// TwinCAT 3 PLC project tmo_optics
// Title: lcls-plc-tmo-optics
// Company: SLAC
// ProjectVersion: 0.0.0
// ProgramVersion: 3.1.4026.17
// CompilerDefines: K
// libraries:
//   LCLS General, * (SLAC)
//   lcls-twincat-common-components, * (SLAC)
//   lcls-twincat-optics, * (SLAC)
//   Tc2_MC2, * (Beckhoff Automation GmbH)
//   Tc2_SerialCom, * (Beckhoff Automation GmbH)
//   Tc2_Standard, * (Beckhoff Automation GmbH)
//   Tc2_System, * (Beckhoff Automation GmbH)
//   Tc2_Utilities, * (Beckhoff Automation GmbH)
//   Tc3_Module, * (Beckhoff Automation GmbH)
//   TcUnit, * (www.tcunit.org)
//   lcls-twincat-motion,4.2.0,SLAC
//   PMPS,3.4.1,SLAC - LCLS
// project tree:
//   DUTs/ ENUM_Si_B4C_Coating_States.TcDUT, E_HomeState.TcDUT (not stored)
//   GVLs/ GVL_COM_Buffers.TcGVL, GVL_M1K4.TcGVL, GVL_M1K4_Constants.TcGVL, GVL_M2K4_RTD.TcGVL, GVL_M2K4_Constants.TcGVL, GVL_M3K4_RTD.TcGVL, GVL_M3K4_Constants.TcGVL, GVL_M4K4_RTD.TcGVL, GVL_M5K4_RTD.TcGVL, GVL_PMPS.TcGVL, GVL_SerialIO.TcGVL
//   / PiezoDriver.TcTTO (not stored), PlcTask.TcTTO, SerialIO.TcTTO (not stored)
//   POUs/ FB_Offset_Coating_States.TcPOU, FB_KBO_Coating_States.TcPOU, Main.TcPOU, PRG_1_PlcTask.TcPOU, PRG_Environment.TcPOU, PRG_MR1K4_SOMS.TcPOU, PRG_MR2K4_KBO.TcPOU, PRG_MR3K4_KBO.TcPOU, PRG_MR4K4_KBO.TcPOU, PRG_MR5K4_KBO.TcPOU, PRG_PMPS.TcPOU, PRG_SL2K4_SCATTER.TcPOU, PRG_States.TcPOU, P_StripeProtections.TcPOU
//   POUs/Serial Comm/ PiezoSerial.TcPOU, P_Serial_Com.TcPOU
//   POUs/temp/ FB_SLITS.TcPOU
// real-time tasks:
//   TASK PlcTask: cycle T#10ms, priority 20, ADS port 350
//   TASK PiezoDriver: cycle T#1ms, priority 3, ADS port 351
//   TASK SerialIO: cycle T#2ms, priority 1, ADS port 352
// motion (NC):
//   TASK NC-Task 1 SAF: cycle T#2ms, priority 4, ADS port 501
//   TASK NC-Task 1 SVB: cycle T#10ms, priority 8, ADS port 511
//   AXIS M1K4-Yup (id 1)
//   AXIS M1K4-Ydwn (id 2)
//   AXIS M1K4-Xup (id 3)
//     General: UnitName=um
//     Dynamic: Acceleration=2000, Deceleration=2000, DelayTime=0.008
//     Velo: Maximum=1000
//     OtherSettings: AllowMotionCmdToSlave=true
//     encoder EncType=29
//       EncPara: ScaleFactorNumerator=0.001, Offset=-24000.3, MaxCount=#xffffffff
//         SoftEndMinControl: Enable=true, Range=-1500
//         SoftEndMaxControl: Enable=true, Range=1500
//         Inc: RefSoftSyncMask=#x0000ffff
//     drive DrvType=24
//       Analog: VeloReferenz=1220.703125, ScaleFactorActTorque=0.1
//       TimeComp: TaskDelayCycles=1
//     controller CtrType=2
//       CtrPara: PriorControlFactor=1
//         PosDiffControl: Range=100
//         PID: PosKp=50, PosExtKp=50, DeadBandPosition=0.4
//         Observer: BandWidth=20
//   AXIS M1K4-Xdwn (id 4)
//     General: UnitName=um
//     Dynamic: Acceleration=2000, Deceleration=2000, DelayTime=0.008
//     Velo: Maximum=1000
//     OtherSettings: AllowMotionCmdToSlave=true
//     encoder EncType=29
//       EncPara: ScaleFactorNumerator=0.001, Offset=-23999.4, MaxCount=#xffffffff
//         SoftEndMinControl: Enable=true, Range=-2000
//         SoftEndMaxControl: Enable=true, Range=2048.5
//         Inc: RefSoftSyncMask=#x0000ffff
//     drive DrvType=24
//       DrvPara: Inverse=true
//         Analog: VeloReferenz=1220.703125, ScaleFactorActTorque=0.1
//         TimeComp: TaskDelayCycles=1
//     controller CtrType=2
//       CtrPara: PriorControlFactor=1
//         PosDiffControl: Range=100
//         PID: PosKp=50, PosExtKp=50, DeadBandPosition=0.4
//         Observer: BandWidth=20
//   AXIS M1K4-Pitch (id 5)
//     General: UnitName=urad
//     Dynamic: Acceleration=390, Deceleration=390, DelayTime=0.008
//     Velo: Maximum=150
//     OtherSettings: AllowMotionCmdToSlave=true
//     encoder EncType=29
//       EncPara: ScaleFactorNumerator=0.001949317739, Offset=-19509, MaxCount=#xffffffff
//         FilterTime: TPos=0.2
//         SoftEndMinControl: Enable=true, Range=-60
//         SoftEndMaxControl: Enable=true, Range=180
//         Inc: RefSoftSyncMask=#x0000ffff
//     drive DrvType=24
//       Analog: VeloReferenz=371.8, ScaleFactorActTorque=0.1
//       TimeComp: TaskDelayCycles=1
//     controller CtrType=2
//       CtrPara: PriorControlFactor=1
//         PosDiffControl: Range=150
//         PID: PosKp=2, PosExtKp=1, DeadBandPosition=0.01
//         Observer: BandWidth=20
//   AXIS M1K4-Bender (id 6)
//     General: UnitName=um
//     Dynamic: Acceleration=100, Deceleration=100, DelayTime=0.008
//     Velo: Maximum=150
//     OtherSettings: AllowMotionCmdToSlave=true
//     encoder EncType=29
//       EncPara: ScaleFactorNumerator=0.001, MaxCount=#xffffffff
//         Inc: RefSoftSyncMask=#x0000ffff
//     drive DrvType=24
//       Analog: VeloReferenz=195.3125, ScaleFactorActTorque=0.1
//       TimeComp: TaskDelayCycles=1
//     controller CtrType=2
//       CtrPara: PriorControlFactor=1
//         PID: PosKp=10, PosExtKp=1, DeadBandPosition=0.04
//         Observer: BandWidth=20
//   AXIS M2K4-X (id 7)
//     Dynamic: AccelerationMaximum=100, DecelerationMaximum=100, Acceleration=100, Deceleration=100, DelayTime=0.008
//     Velo: Maximum=20
//     OtherSettings: AllowMotionCmdToSlave=true
//     encoder EncType=29
//       EncPara: ScaleFactorNumerator=5e-06, Offset=-30.6825, MaxCount=#xffffffff, ReferenceSystem=1
//         SoftEndMinControl: Enable=true, Range=0.2
//         SoftEndMaxControl: Enable=true, Range=2.1
//         Inc: RefSoftSyncMask=#x0000ffff
//     drive DrvType=24
//       DrvPara: Inverse=true
//         Analog: VeloReferenz=20, ScaleFactorActTorque=0.1
//         TimeComp: TaskDelayCycles=1
//     controller CtrType=2
//       CtrPara: PriorControlFactor=1
//         PosDiffControl: Range=0.1
//         PID: DeadBandPosition=0.001
//         Observer: BandWidth=20
//   AXIS M2K4-Y (id 8)
//     Dynamic: AccelerationMaximum=10, DecelerationMaximum=10, Acceleration=10, Deceleration=10, Jerk=15, DelayTime=0.008
//     Velo: Maximum=1.25
//     OtherSettings: AllowMotionCmdToSlave=true
//     encoder EncType=29
//       EncPara: ScaleFactorNumerator=5e-06, Offset=-30.18, MaxCount=#xffffffff, ReferenceSystem=1
//         SoftEndMinControl: Enable=true, Range=-12.5
//         SoftEndMaxControl: Enable=true, Range=13.39
//         Inc: RefSoftSyncMask=#x0000ffff
//     drive DrvType=24
//       DrvPara: Inverse=true
//         Analog: VeloReferenz=1.25, ScaleFactorActTorque=0.1
//         TimeComp: TaskDelayCycles=1
//     controller CtrType=2
//       CtrPara: PriorControlFactor=1
//         PosDiffControl: Range=0.1
//         PID: DeadBandPosition=0.001
//         Observer: BandWidth=20
//   AXIS M2K4-rY (id 9)
//     General: UnitName=urad
//     Dynamic: AccelerationMaximum=400, DecelerationMaximum=400, Acceleration=400, Deceleration=400, Jerk=1200, DelayTime=0.008
//     Velo: Maximum=166.67
//     OtherSettings: AllowMotionCmdToSlave=true
//     encoder EncType=29
//       EncPara: ScaleFactorNumerator=0.005348, Offset=-194502.025, MaxCount=#xffffffff, ReferenceSystem=1
//         FilterTime: TPos=0.01
//         SoftEndMinControl: Enable=true, Range=14370
//         SoftEndMaxControl: Enable=true, Range=14850
//         Inc: RefSoftSyncMask=#x0000ffff
//     drive DrvType=24
//       Analog: VeloReferenz=166.67, ScaleFactorActTorque=0.1
//       TimeComp: TaskDelayCycles=1
//     controller CtrType=2
//       CtrPara: PriorControlFactor=1
//         PosDiffControl: Range=40
//         PID: PosKp=0.5, DeadBandPosition=0.01
//         Observer: BandWidth=20
//   AXIS M2K4-BEND-US (id 10)
//     Dynamic: AccelerationMaximum=0.6, DecelerationMaximum=0.6, Acceleration=0.6, Deceleration=0.6, Jerk=1.2, DelayTime=0.008
//     Velo: Maximum=0.1
//     OtherSettings: AllowMotionCmdToSlave=true
//     encoder EncType=29
//       EncPara: ScaleFactorNumerator=1e-06, MaxCount=#xffffffff, ReferenceSystem=1
//         SoftEndMinControl: Enable=true, Range=6.4549
//         SoftEndMaxControl: Enable=true, Range=16.0941
//         Inc: RefSoftSyncMask=#x0000ffff
//     drive DrvType=24
//       DrvPara: Inverse=true
//         Analog: VeloReferenz=0.1, ScaleFactorActTorque=0.1
//         TimeComp: TaskDelayCycles=1
//     controller CtrType=2
//       CtrPara: PriorControlFactor=1
//         PosDiffControl: Range=0.2
//         PID: PosKp=15, PosExtKp=1, DeadBandPosition=0.0002
//         Observer: BandWidth=20
//   AXIS M2K4-BEND-DS (id 11)
//     Dynamic: AccelerationMaximum=0.6, DecelerationMaximum=0.6, Acceleration=0.6, Deceleration=0.6, Jerk=1.2, DelayTime=0.008
//     Velo: Maximum=0.1
//     OtherSettings: AllowMotionCmdToSlave=true
//     encoder EncType=29
//       EncPara: ScaleFactorNumerator=1e-06, MaxCount=#xffffffff, ReferenceSystem=1
//         SoftEndMinControl: Enable=true, Range=10.5742
//         SoftEndMaxControl: Enable=true, Range=22.2169
//         Inc: RefSoftSyncMask=#x0000ffff
//     drive DrvType=24
//       DrvPara: Inverse=true
//         Analog: VeloReferenz=0.1, ScaleFactorActTorque=0.1
//         TimeComp: TaskDelayCycles=1
//     controller CtrType=2
//       CtrPara: PriorControlFactor=1
//         PosDiffControl: Range=0.2
//         PID: PosKp=15, PosExtKp=1, DeadBandPosition=0.0002
//         Observer: BandWidth=20
//   AXIS M3K4-X (id 12)
//     Dynamic: AccelerationMaximum=100, DecelerationMaximum=100, Acceleration=100, Deceleration=100, DelayTime=0.008
//     Velo: Maximum=20
//     OtherSettings: AllowMotionCmdToSlave=true
//     encoder EncType=29
//       EncPara: ScaleFactorNumerator=5e-06, Offset=-31.1, MaxCount=#xffffffff, ReferenceSystem=1
//         SoftEndMinControl: Enable=true, Range=-10.179
//         SoftEndMaxControl: Enable=true, Range=12.0995
//         Inc: RefSoftSyncMask=#x0000ffff
//     drive DrvType=24
//       DrvPara: Inverse=true
//         Analog: VeloReferenz=20, ScaleFactorActTorque=0.1
//         TimeComp: TaskDelayCycles=1
//     controller CtrType=2
//       CtrPara: PriorControlFactor=1
//         PosDiffControl: Range=0.1
//         PID: DeadBandPosition=0.001
//         Observer: BandWidth=20
//   AXIS M3K4-Y (id 13)
//     Dynamic: AccelerationMaximum=10, DecelerationMaximum=10, Acceleration=10, Deceleration=10, Jerk=15, DelayTime=0.008
//     Velo: Maximum=1.25
//     OtherSettings: AllowMotionCmdToSlave=true
//     encoder EncType=29
//       EncPara: ScaleFactorNumerator=5e-06, Offset=-29.68, MaxCount=#xffffffff, ReferenceSystem=1
//         SoftEndMinControl: Enable=true, Range=0.25
//         SoftEndMaxControl: Enable=true, Range=2.15
//         Inc: RefSoftSyncMask=#x0000ffff
//     drive DrvType=24
//       DrvPara: Inverse=true
//         Analog: VeloReferenz=1.25, ScaleFactorActTorque=0.1
//         TimeComp: TaskDelayCycles=1
//     controller CtrType=2
//       CtrPara: PriorControlFactor=1
//         PosDiffControl: Range=0.1
//         PID: DeadBandPosition=0.001
//         Observer: BandWidth=20
//   AXIS M3K4-rX (id 14)
//     General: UnitName=urad
//     Dynamic: AccelerationMaximum=300, DecelerationMaximum=300, Acceleration=300, Deceleration=300, Jerk=900, DelayTime=0.008
//     Velo: Maximum=140.84
//     OtherSettings: AllowMotionCmdToSlave=true
//     encoder EncType=29
//       EncPara: ScaleFactorNumerator=0.002577, Offset=-136547, MaxCount=#xffffffff, ReferenceSystem=1
//         FilterTime: TPos=0.01
//         SoftEndMinControl: Enable=true, Range=-12560
//         SoftEndMaxControl: Enable=true, Range=-12090
//         Inc: RefSoftSyncMask=#x0000ffff
//     drive DrvType=24
//       Analog: VeloReferenz=140.84, ScaleFactorActTorque=0.1
//       TimeComp: TaskDelayCycles=1
//     controller CtrType=2
//       CtrPara: PriorControlFactor=1
//         PosDiffControl: Range=10
//         PID: PosKp=0.5, DeadBandPosition=0.01
//         Observer: BandWidth=20
//   AXIS M3K4-BEND-US (id 15)
//     Dynamic: AccelerationMaximum=0.6, DecelerationMaximum=0.6, Acceleration=0.6, Deceleration=0.6, Jerk=1.2, DelayTime=0.008
//     Velo: Maximum=0.1
//     OtherSettings: AllowMotionCmdToSlave=true
//     encoder EncType=29
//       EncPara: ScaleFactorNumerator=1e-06, MaxCount=#xffffffff, ReferenceSystem=1
//         SoftEndMinControl: Enable=true, Range=12.5315
//         SoftEndMaxControl: Enable=true, Range=22.979
//         Inc: RefSoftSyncMask=#x0000ffff
//     drive DrvType=24
//       DrvPara: Inverse=true
//         Analog: VeloReferenz=0.1, ScaleFactorActTorque=0.1
//         TimeComp: TaskDelayCycles=1
//     controller CtrType=2
//       CtrPara: PriorControlFactor=1
//         PosDiffControl: Range=0.2
//         PID: PosKp=15, PosExtKp=1, DeadBandPosition=0.0002
//         Observer: BandWidth=20
//   AXIS M3K4-BEND-DS (id 16)
//     Dynamic: AccelerationMaximum=0.6, DecelerationMaximum=0.6, Acceleration=0.6, Deceleration=0.6, Jerk=1.2, DelayTime=0.008
//     Velo: Maximum=0.1
//     OtherSettings: AllowMotionCmdToSlave=true
//     encoder EncType=29
//       EncPara: ScaleFactorNumerator=1e-06, MaxCount=#xffffffff, ReferenceSystem=1
//         SoftEndMinControl: Enable=true, Range=8.0419
//         SoftEndMaxControl: Enable=true, Range=22.8443
//         Inc: RefSoftSyncMask=#x0000ffff
//     drive DrvType=24
//       DrvPara: Inverse=true
//         Analog: VeloReferenz=0.1, ScaleFactorActTorque=0.1
//         TimeComp: TaskDelayCycles=1
//     controller CtrType=2
//       CtrPara: PriorControlFactor=1
//         PosDiffControl: Range=0.2
//         PID: PosKp=15, PosExtKp=1, DeadBandPosition=0.0002
//         Observer: BandWidth=20
//   AXIS M4K4 X (id 17)
//     Dynamic: AccelerationMaximum=100, DecelerationMaximum=100, Acceleration=100, Deceleration=100, DelayTime=0.008
//     Velo: Maximum=0.3
//     OtherSettings: AllowMotionCmdToSlave=true
//     encoder EncType=29
//       EncPara: ScaleFactorNumerator=5e-06, Offset=-28.961399, MaxCount=#xffffffff, ReferenceSystem=1
//         SoftEndMinControl: Range=-11.2
//         SoftEndMaxControl: Range=13.2
//         Inc: RefSoftSyncMask=#x0000ffff
//     drive DrvType=24
//       DrvPara: Inverse=true
//         Analog: VeloReferenz=20, ScaleFactorActTorque=0.1
//         TimeComp: TaskDelayCycles=1
//     controller CtrType=2
//       CtrPara: PriorControlFactor=1
//         PosDiffControl: Range=0.2
//         PID: DeadBandPosition=0.001
//         Observer: BandWidth=20
//   AXIS M4K4 Y (id 18)
//     Dynamic: AccelerationMaximum=100, DecelerationMaximum=100, Acceleration=100, Deceleration=100, DelayTime=0.008
//     Velo: Maximum=0.2
//     OtherSettings: AllowMotionCmdToSlave=true
//     encoder EncType=29
//       EncPara: ScaleFactorNumerator=5e-06, Offset=-30.3992, MaxCount=#xffffffff, ReferenceSystem=1
//         SoftEndMinControl: Enable=true, Range=-0.5
//         SoftEndMaxControl: Enable=true, Range=1.25
//         Inc: RefSoftSyncMask=#x0000ffff
//     drive DrvType=24
//       DrvPara: Inverse=true
//         Analog: VeloReferenz=1.25, ScaleFactorActTorque=0.1
//         TimeComp: TaskDelayCycles=1
//     controller CtrType=2
//       CtrPara: PriorControlFactor=1
//         PosDiffControl: Range=0.2
//         PID: PosKp=3, DeadBandPosition=0.001
//         Observer: BandWidth=20
//   AXIS M4K4 Z (id 19)
//     Dynamic: AccelerationMaximum=100, DecelerationMaximum=100, Acceleration=100, Deceleration=100, DelayTime=0.008
//     Velo: Maximum=0.2
//     OtherSettings: AllowMotionCmdToSlave=true
//     encoder EncType=29
//       EncPara: ScaleFactorNumerator=5e-06, Offset=-21445.3535, MaxCount=#xffffffff, ReferenceSystem=1
//         SoftEndMinControl: Enable=true, Range=-1.5
//         SoftEndMaxControl: Enable=true, Range=0.85
//         Inc: RefSoftSyncMask=#x0000ffff
//     drive DrvType=24
//       DrvPara: Inverse=true
//         Analog: VeloReferenz=1.25, ScaleFactorActTorque=0.1
//         TimeComp: TaskDelayCycles=1
//     controller CtrType=2
//       CtrPara: PriorControlFactor=1
//         PosDiffControl: Range=0.2
//         PID: PosKp=2, DeadBandPosition=0.01
//         Observer: BandWidth=20
//   AXIS M4K4 rX (id 20)
//     General: UnitName=urad
//     Dynamic: AccelerationMaximum=100, DecelerationMaximum=100, Acceleration=100, Deceleration=100, DelayTime=0.008
//     Velo: Maximum=50
//     OtherSettings: AllowMotionCmdToSlave=true
//     encoder EncType=29
//       EncPara: ScaleFactorNumerator=0.0025826, Offset=-132192.8499, MaxCount=#xffffffff, ReferenceSystem=1
//         FilterTime: TPos=0.2
//         SoftEndMinControl: Enable=true, Range=-300
//         SoftEndMaxControl: Enable=true, Range=35
//         Inc: RefSoftSyncMask=#x0000ffff
//     drive DrvType=24
//       Analog: VeloReferenz=140.69, ScaleFactorActTorque=0.1
//       TimeComp: TaskDelayCycles=1
//     controller CtrType=2
//       CtrPara: PriorControlFactor=1
//         PosDiffControl: Range=10
//         PID: PosExtKp=4, DeadBandPosition=0.01
//         Observer: BandWidth=20
//   AXIS M5K4 X (id 21)
//     Dynamic: AccelerationMaximum=100, DecelerationMaximum=100, Acceleration=100, Deceleration=100, DelayTime=0.008
//     Velo: Maximum=0.2
//     OtherSettings: AllowMotionCmdToSlave=true
//     encoder EncType=29
//       EncPara: ScaleFactorNumerator=5e-06, Offset=-29.80379, MaxCount=#xffffffff, ReferenceSystem=1
//         SoftEndMinControl: Enable=true, Range=-2.3
//         SoftEndMaxControl: Enable=true, Range=-0.37
//         Inc: RefSoftSyncMask=#x0000ffff
//     drive DrvType=24
//       DrvPara: Inverse=true
//         Analog: VeloReferenz=20, ScaleFactorActTorque=0.1
//         TimeComp: TaskDelayCycles=1
//     controller CtrType=2
//       CtrPara: PriorControlFactor=1
//         PosDiffControl: Range=0.2
//         PID: DeadBandPosition=0.001
//         Observer: BandWidth=20
//   AXIS M5K4 Y (id 22)
//     Dynamic: AccelerationMaximum=100, DecelerationMaximum=100, Acceleration=100, Deceleration=100, DelayTime=0.008
//     Velo: Maximum=0.3
//     OtherSettings: AllowMotionCmdToSlave=true
//     encoder EncType=29
//       EncPara: ScaleFactorNumerator=5e-06, Offset=-29.7766, MaxCount=#xffffffff, ReferenceSystem=1
//         SoftEndMinControl: Range=-12.3
//         SoftEndMaxControl: Range=12.33
//         Inc: RefSoftSyncMask=#x0000ffff
//     drive DrvType=24
//       DrvPara: Inverse=true
//         Analog: VeloReferenz=1.25, ScaleFactorActTorque=0.1
//         TimeComp: TaskDelayCycles=1
//     controller CtrType=2
//       CtrPara: PriorControlFactor=1
//         PosDiffControl: Range=0.2
//         PID: DeadBandPosition=0.001
//         Observer: BandWidth=20
//   AXIS M5K4 Z (id 23)
//     Dynamic: AccelerationMaximum=100, DecelerationMaximum=100, Acceleration=100, Deceleration=100, DelayTime=0.008
//     Velo: Maximum=0.2
//     OtherSettings: AllowMotionCmdToSlave=true
//     encoder EncType=29
//       EncPara: ScaleFactorNumerator=5e-06, Offset=-21444.5039, MaxCount=#xffffffff, ReferenceSystem=1
//         SoftEndMinControl: Enable=true, Range=-0.69
//         SoftEndMaxControl: Enable=true, Range=1.02
//         Inc: RefSoftSyncMask=#x0000ffff
//     drive DrvType=24
//       DrvPara: Inverse=true
//         Analog: VeloReferenz=1.25, ScaleFactorActTorque=0.1
//         TimeComp: TaskDelayCycles=1
//     controller CtrType=2
//       CtrPara: PriorControlFactor=1
//         PosDiffControl: Range=0.2
//         PID: PosExtVelo=1, DeadBandPosition=0.01
//         Observer: BandWidth=20
//   AXIS M5K4 rY (id 24)
//     General: UnitName=urad
//     Dynamic: AccelerationMaximum=100, DecelerationMaximum=100, Acceleration=100, Deceleration=100, DelayTime=0.008
//     Velo: Maximum=50
//     OtherSettings: AllowMotionCmdToSlave=true
//     encoder EncType=29
//       EncPara: ScaleFactorNumerator=0.00504, Offset=-198169.78, MaxCount=#xffffffff, ReferenceSystem=1
//         FilterTime: TPos=0.2
//         SoftEndMinControl: Enable=true, Range=-260
//         SoftEndMaxControl: Enable=true, Range=200
//         Inc: RefSoftSyncMask=#x0000ffff
//     drive DrvType=24
//       Analog: VeloReferenz=192.31, ScaleFactorActTorque=0.1
//       TimeComp: TaskDelayCycles=1
//     controller CtrType=2
//       CtrPara: PriorControlFactor=1
//         PosDiffControl: Range=10
//         PID: PosKp=2, PosExtKp=10, DeadBandPosition=0.01
//         Observer: BandWidth=20
//   AXIS SL2K4_TOP (id 25)
//     Dynamic: AccelerationMaximum=0.25, DecelerationMaximum=0.25, Acceleration=0.25, Deceleration=0.25, Jerk=0.4
//     Velo: RefSearch=0.05, RefSync=0.025, SlowManual=0.1, FastManual=0.1, Fast=3, Maximum=0.5
//     PositionAreaControl: Enable=false
//     TargetPosControl: Range=0.01
//     OtherSettings: AllowMotionCmdToSlave=true, PulseDistancePos=0.005, PulseDistanceNeg=0.005
//     encoder EncType=4
//       EncPara: ScaleFactorNumerator=1e-06, Inverse=true, MaxCount=#xffffffff
//         SoftEndMinControl: Enable=true, Range=-0.1
//         SoftEndMaxControl: Enable=true, Range=4.35
//         Inc: RefSoftSyncMask=#x0000ffff
//     drive DrvType=24
//       DrvPara: Inverse=true
//         Analog: VeloReferenz=3, TorqueSetpointScale=10, ScaleFactorActTorque=0.1
//         TimeComp: TaskDelayCycles=1
//     controller CtrType=1
//       CtrPara: PriorControlFactor=1
//         PosDiffControl: Range=0.2
//         Observer: BandWidth=20
//   AXIS SL2K4_BOTTOM (id 26)
//     Dynamic: AccelerationMaximum=0.25, DecelerationMaximum=0.25, Acceleration=0.25, Deceleration=0.25, Jerk=0.4
//     Velo: RefSearch=0.05, RefSync=0.025, SlowManual=0.1, FastManual=0.1, Maximum=0.5
//     PositionAreaControl: Enable=false
//     TargetPosControl: Range=0.01
//     OtherSettings: AllowMotionCmdToSlave=true, PulseDistancePos=0.005, PulseDistanceNeg=0.005
//     encoder EncType=4
//       EncPara: ScaleFactorNumerator=1e-06, MaxCount=#xffffffff
//         SoftEndMinControl: Enable=true, Range=-4.6
//         SoftEndMaxControl: Enable=true, Range=-0.4
//         Inc: RefSoftSyncMask=#x0000ffff
//     drive DrvType=24
//       Analog: VeloReferenz=3, TorqueSetpointScale=10, ScaleFactorActTorque=0.1
//       TimeComp: TaskDelayCycles=1
//     controller CtrType=1
//       CtrPara: PriorControlFactor=1
//         PosDiffControl: Range=0.2
//         Observer: BandWidth=20
//   AXIS SL2K4_NORTH (id 27)
//     Dynamic: AccelerationMaximum=0.25, DecelerationMaximum=0.25, Acceleration=0.25, Deceleration=0.25, Jerk=0.4
//     Velo: RefSearch=0.05, RefSync=0.025, SlowManual=0.1, FastManual=0.1, Maximum=0.5
//     OtherSettings: AllowMotionCmdToSlave=true, PulseDistancePos=0.005, PulseDistanceNeg=0.005
//     encoder EncType=4
//       EncPara: ScaleFactorNumerator=1e-06, Inverse=true, MaxCount=#xffffffff
//         SoftEndMinControl: Enable=true, Range=0.3
//         SoftEndMaxControl: Enable=true, Range=4.35
//         Inc: RefSoftSyncMask=#x0000ffff
//     drive DrvType=24
//       DrvPara: Inverse=true
//         Analog: VeloReferenz=3, TorqueSetpointScale=10, ScaleFactorActTorque=0.1
//         TimeComp: TaskDelayCycles=1
//     controller CtrType=1
//       CtrPara: PriorControlFactor=1
//         PosDiffControl: Range=0.2
//         Observer: BandWidth=20
//   AXIS SL2K4_SOUTH (id 28)
//     Dynamic: AccelerationMaximum=0.25, DecelerationMaximum=0.25, Acceleration=0.25, Deceleration=0.25, Jerk=0.4
//     Velo: RefSearch=0.05, RefSync=0.025, SlowManual=0.1, FastManual=0.1, Maximum=0.5
//     TargetPosControl: Range=0.01
//     OtherSettings: AllowMotionCmdToSlave=true, PulseDistancePos=0.005, PulseDistanceNeg=0.005
//     encoder EncType=4
//       EncPara: ScaleFactorNumerator=1e-06, MaxCount=#xffffffff
//         SoftEndMinControl: Enable=true, Range=-4.5
//         SoftEndMaxControl: Enable=true, Range=-0.3
//         Inc: RefSoftSyncMask=#x0000ffff
//     drive DrvType=24
//       Analog: VeloReferenz=3, TorqueSetpointScale=10, ScaleFactorActTorque=0.1
//       TimeComp: TaskDelayCycles=1
//     controller CtrType=1
//       CtrPara: PriorControlFactor=1
//         PosDiffControl: Range=0.2
//         Observer: BandWidth=20
// I/O:
//   DEVICE Device 1 (EtherCAT), AmsNetId 172.21.92.63.2.1
//     Term 1 (EK1200)
// variable links:
//   Axes/M4K4 X <-> Device 1 (EtherCAT)/Term 1 (EK1200)/Term 39 (EK1122)/Term 94 (EK1100)/EL5042_M4K4X_M4K4Y
//     Enc/Inputs/In/nComState @bit 1 <-> WcState/InputToggle
//     Enc/Inputs/In/nComState <-> WcState/WcState
//     Enc/Inputs/In/nDataIn1 <-> FB Inputs Channel 1/Position
//     Enc/Inputs/In/nState1 @bit 12 <-> FB Inputs Channel 1/Status/Diag
//     Enc/Inputs/In/nState1 @bit 1 <-> FB Inputs Channel 1/Status/Error
//     Enc/Inputs/In/nState1 @bit 14 <-> FB Inputs Channel 1/Status/Input cycle counter
//     Enc/Inputs/In/nState1 @bit 2 <-> FB Inputs Channel 1/Status/Ready
//     Enc/Inputs/In/nState1 @bit 13 <-> FB Inputs Channel 1/Status/TxPDO State
//     Enc/Inputs/In/nState1 <-> FB Inputs Channel 1/Status/Warning
//   Axes/M4K4 X <-> Device 1 (EtherCAT)/Term 1 (EK1200)/Term 39 (EK1122)/Term 94 (EK1100)/EL7041-0052_M4K4X
//     Drive/Inputs/In/nState1 @bit 3 <-> STM Status/Status/Error
//     Drive/Inputs/In/nState1 @bit 5 <-> STM Status/Status/Moving negative
//     Drive/Inputs/In/nState1 @bit 4 <-> STM Status/Status/Moving positive
//     Drive/Inputs/In/nState1 @bit 1 <-> STM Status/Status/Ready
//     Drive/Inputs/In/nState1 <-> STM Status/Status/Ready to enable
//     Drive/Inputs/In/nState1 @bit 6 <-> STM Status/Status/Torque reduced
//     Drive/Inputs/In/nState1 @bit 2 <-> STM Status/Status/Warning
//     Drive/Inputs/In/nState2 @bit 3 <-> STM Status/Status/Digital input 1
//     Drive/Inputs/In/nState2 @bit 4 <-> STM Status/Status/Digital input 2
//     Drive/Inputs/In/nState2 @bit 5 <-> STM Status/Status/Sync error
//     Drive/Inputs/In/nState2 @bit 7 <-> STM Status/Status/TxPDO Toggle
//     Drive/Inputs/In/nState4 @bit 1 <-> WcState/InputToggle
//     Drive/Inputs/In/nState4 <-> WcState/WcState
//     Drive/Outputs/Out/nCtrl1 <-> STM Control/Control/Enable
//     Drive/Outputs/Out/nCtrl1 @bit 2 <-> STM Control/Control/Reduce torque
//     Drive/Outputs/Out/nCtrl1 @bit 1 <-> STM Control/Control/Reset
//     Drive/Outputs/Out/nDataOut2[0] <-> STM Velocity/Velocity
//   Axes/M4K4 Y <-> Device 1 (EtherCAT)/Term 1 (EK1200)/Term 39 (EK1122)/Term 94 (EK1100)/EL5042_M4K4X_M4K4Y
//     Enc/Inputs/In/nComState @bit 1 <-> WcState/InputToggle
//     Enc/Inputs/In/nComState <-> WcState/WcState
//     Enc/Inputs/In/nDataIn1 <-> FB Inputs Channel 2/Position
//     Enc/Inputs/In/nState1 @bit 12 <-> FB Inputs Channel 2/Status/Diag
//     Enc/Inputs/In/nState1 @bit 1 <-> FB Inputs Channel 2/Status/Error
//     Enc/Inputs/In/nState1 @bit 14 <-> FB Inputs Channel 2/Status/Input cycle counter
//     Enc/Inputs/In/nState1 @bit 2 <-> FB Inputs Channel 2/Status/Ready
//     Enc/Inputs/In/nState1 @bit 13 <-> FB Inputs Channel 2/Status/TxPDO State
//     Enc/Inputs/In/nState1 <-> FB Inputs Channel 2/Status/Warning
//   Axes/M4K4 Y <-> Device 1 (EtherCAT)/Term 1 (EK1200)/Term 39 (EK1122)/Term 94 (EK1100)/EL7041-0052_M4K4Y
//     Drive/Inputs/In/nState1 @bit 3 <-> STM Status/Status/Error
//     Drive/Inputs/In/nState1 @bit 5 <-> STM Status/Status/Moving negative
//     Drive/Inputs/In/nState1 @bit 4 <-> STM Status/Status/Moving positive
//     Drive/Inputs/In/nState1 @bit 1 <-> STM Status/Status/Ready
//     Drive/Inputs/In/nState1 <-> STM Status/Status/Ready to enable
//     Drive/Inputs/In/nState1 @bit 6 <-> STM Status/Status/Torque reduced
//     Drive/Inputs/In/nState1 @bit 2 <-> STM Status/Status/Warning
//     Drive/Inputs/In/nState2 @bit 3 <-> STM Status/Status/Digital input 1
//     Drive/Inputs/In/nState2 @bit 4 <-> STM Status/Status/Digital input 2
//     Drive/Inputs/In/nState2 @bit 5 <-> STM Status/Status/Sync error
//     Drive/Inputs/In/nState2 @bit 7 <-> STM Status/Status/TxPDO Toggle
//     Drive/Inputs/In/nState4 @bit 1 <-> WcState/InputToggle
//     Drive/Inputs/In/nState4 <-> WcState/WcState
//     Drive/Outputs/Out/nCtrl1 <-> STM Control/Control/Enable
//     Drive/Outputs/Out/nCtrl1 @bit 2 <-> STM Control/Control/Reduce torque
//     Drive/Outputs/Out/nCtrl1 @bit 1 <-> STM Control/Control/Reset
//     Drive/Outputs/Out/nDataOut2[0] <-> STM Velocity/Velocity
//   Axes/M4K4 Z <-> Device 1 (EtherCAT)/Term 1 (EK1200)/Term 39 (EK1122)/Term 94 (EK1100)/EL5042_M4K4Z_M4K4rX
//     Enc/Inputs/In/nComState @bit 1 <-> WcState/InputToggle
//     Enc/Inputs/In/nComState <-> WcState/WcState
//     Enc/Inputs/In/nDataIn1 <-> FB Inputs Channel 1/Position
//     Enc/Inputs/In/nState1 @bit 12 <-> FB Inputs Channel 1/Status/Diag
//     Enc/Inputs/In/nState1 @bit 1 <-> FB Inputs Channel 1/Status/Error
//     Enc/Inputs/In/nState1 @bit 14 <-> FB Inputs Channel 1/Status/Input cycle counter
//     Enc/Inputs/In/nState1 @bit 2 <-> FB Inputs Channel 1/Status/Ready
//     Enc/Inputs/In/nState1 @bit 13 <-> FB Inputs Channel 1/Status/TxPDO State
//     Enc/Inputs/In/nState1 <-> FB Inputs Channel 1/Status/Warning
//   Axes/M4K4 Z <-> Device 1 (EtherCAT)/Term 1 (EK1200)/Term 39 (EK1122)/Term 94 (EK1100)/EL7041-0052_M4K4Z
//     Drive/Inputs/In/nState1 @bit 3 <-> STM Status/Status/Error
//     Drive/Inputs/In/nState1 @bit 5 <-> STM Status/Status/Moving negative
//     Drive/Inputs/In/nState1 @bit 4 <-> STM Status/Status/Moving positive
//     Drive/Inputs/In/nState1 @bit 1 <-> STM Status/Status/Ready
//     Drive/Inputs/In/nState1 <-> STM Status/Status/Ready to enable
//     Drive/Inputs/In/nState1 @bit 6 <-> STM Status/Status/Torque reduced
//     Drive/Inputs/In/nState1 @bit 2 <-> STM Status/Status/Warning
//     Drive/Inputs/In/nState2 @bit 3 <-> STM Status/Status/Digital input 1
//     Drive/Inputs/In/nState2 @bit 4 <-> STM Status/Status/Digital input 2
//     Drive/Inputs/In/nState2 @bit 5 <-> STM Status/Status/Sync error
//     Drive/Inputs/In/nState2 @bit 7 <-> STM Status/Status/TxPDO Toggle
//     Drive/Inputs/In/nState4 @bit 1 <-> WcState/InputToggle
//     Drive/Inputs/In/nState4 <-> WcState/WcState
//     Drive/Outputs/Out/nCtrl1 <-> STM Control/Control/Enable
//     Drive/Outputs/Out/nCtrl1 @bit 2 <-> STM Control/Control/Reduce torque
//     Drive/Outputs/Out/nCtrl1 @bit 1 <-> STM Control/Control/Reset
//     Drive/Outputs/Out/nDataOut2[0] <-> STM Velocity/Velocity
//   Axes/M4K4 rX <-> Device 1 (EtherCAT)/Term 1 (EK1200)/Term 39 (EK1122)/Term 94 (EK1100)/EL5042_M4K4Z_M4K4rX
//     Enc/Inputs/In/nComState @bit 1 <-> WcState/InputToggle
//     Enc/Inputs/In/nComState <-> WcState/WcState
//     Enc/Inputs/In/nDataIn1 <-> FB Inputs Channel 2/Position
//     Enc/Inputs/In/nState1 @bit 12 <-> FB Inputs Channel 2/Status/Diag
//     Enc/Inputs/In/nState1 @bit 1 <-> FB Inputs Channel 2/Status/Error
//     Enc/Inputs/In/nState1 @bit 14 <-> FB Inputs Channel 2/Status/Input cycle counter
//     Enc/Inputs/In/nState1 @bit 2 <-> FB Inputs Channel 2/Status/Ready
//     Enc/Inputs/In/nState1 @bit 13 <-> FB Inputs Channel 2/Status/TxPDO State
//     Enc/Inputs/In/nState1 <-> FB Inputs Channel 2/Status/Warning
//   Axes/M4K4 rX <-> Device 1 (EtherCAT)/Term 1 (EK1200)/Term 39 (EK1122)/Term 94 (EK1100)/EL7041-0052_M4K4rX
//     Drive/Inputs/In/nState1 @bit 3 <-> STM Status/Status/Error
//     Drive/Inputs/In/nState1 @bit 5 <-> STM Status/Status/Moving negative
//     Drive/Inputs/In/nState1 @bit 4 <-> STM Status/Status/Moving positive
//     Drive/Inputs/In/nState1 @bit 1 <-> STM Status/Status/Ready
//     Drive/Inputs/In/nState1 <-> STM Status/Status/Ready to enable
//     Drive/Inputs/In/nState1 @bit 6 <-> STM Status/Status/Torque reduced
//     Drive/Inputs/In/nState1 @bit 2 <-> STM Status/Status/Warning
//     Drive/Inputs/In/nState2 @bit 3 <-> STM Status/Status/Digital input 1
//     Drive/Inputs/In/nState2 @bit 4 <-> STM Status/Status/Digital input 2
//     Drive/Inputs/In/nState2 @bit 5 <-> STM Status/Status/Sync error
//     Drive/Inputs/In/nState2 @bit 7 <-> STM Status/Status/TxPDO Toggle
//     Drive/Inputs/In/nState4 @bit 1 <-> WcState/InputToggle
//     Drive/Inputs/In/nState4 <-> WcState/WcState
//     Drive/Outputs/Out/nCtrl1 <-> STM Control/Control/Enable
//     Drive/Outputs/Out/nCtrl1 @bit 2 <-> STM Control/Control/Reduce torque
//     Drive/Outputs/Out/nCtrl1 @bit 1 <-> STM Control/Control/Reset
//     Drive/Outputs/Out/nDataOut2[0] <-> STM Velocity/Velocity
//   Axes/M5K4 X <-> Device 1 (EtherCAT)/Term 1 (EK1200)/Term 39 (EK1122)/Term 94 (EK1100)/EL5042_M5K4X_M5K4Y
//     Enc/Inputs/In/nComState @bit 1 <-> WcState/InputToggle
//     Enc/Inputs/In/nComState <-> WcState/WcState
//     Enc/Inputs/In/nDataIn1 <-> FB Inputs Channel 1/Position
//     Enc/Inputs/In/nState1 @bit 12 <-> FB Inputs Channel 1/Status/Diag
//     Enc/Inputs/In/nState1 @bit 1 <-> FB Inputs Channel 1/Status/Error
//     Enc/Inputs/In/nState1 @bit 14 <-> FB Inputs Channel 1/Status/Input cycle counter
//     Enc/Inputs/In/nState1 @bit 2 <-> FB Inputs Channel 1/Status/Ready
//     Enc/Inputs/In/nState1 @bit 13 <-> FB Inputs Channel 1/Status/TxPDO State
//     Enc/Inputs/In/nState1 <-> FB Inputs Channel 1/Status/Warning
//   Axes/M5K4 X <-> Device 1 (EtherCAT)/Term 1 (EK1200)/Term 39 (EK1122)/Term 94 (EK1100)/EL7041-0052_M5K4X
//     Drive/Inputs/In/nState1 @bit 3 <-> STM Status/Status/Error
//     Drive/Inputs/In/nState1 @bit 5 <-> STM Status/Status/Moving negative
//     Drive/Inputs/In/nState1 @bit 4 <-> STM Status/Status/Moving positive
//     Drive/Inputs/In/nState1 @bit 1 <-> STM Status/Status/Ready
//     Drive/Inputs/In/nState1 <-> STM Status/Status/Ready to enable
//     Drive/Inputs/In/nState1 @bit 6 <-> STM Status/Status/Torque reduced
//     Drive/Inputs/In/nState1 @bit 2 <-> STM Status/Status/Warning
//     Drive/Inputs/In/nState2 @bit 3 <-> STM Status/Status/Digital input 1
//     Drive/Inputs/In/nState2 @bit 4 <-> STM Status/Status/Digital input 2
//     Drive/Inputs/In/nState2 @bit 5 <-> STM Status/Status/Sync error
//     Drive/Inputs/In/nState2 @bit 7 <-> STM Status/Status/TxPDO Toggle
//     Drive/Inputs/In/nState4 @bit 1 <-> WcState/InputToggle
//     Drive/Inputs/In/nState4 <-> WcState/WcState
//     Drive/Outputs/Out/nCtrl1 <-> STM Control/Control/Enable
//     Drive/Outputs/Out/nCtrl1 @bit 2 <-> STM Control/Control/Reduce torque
//     Drive/Outputs/Out/nCtrl1 @bit 1 <-> STM Control/Control/Reset
//     Drive/Outputs/Out/nDataOut2[0] <-> STM Velocity/Velocity
//   Axes/M5K4 Y <-> Device 1 (EtherCAT)/Term 1 (EK1200)/Term 39 (EK1122)/Term 94 (EK1100)/EL5042_M5K4X_M5K4Y
//     Enc/Inputs/In/nComState @bit 1 <-> WcState/InputToggle
//     Enc/Inputs/In/nComState <-> WcState/WcState
//     Enc/Inputs/In/nDataIn1 <-> FB Inputs Channel 2/Position
//     Enc/Inputs/In/nState1 @bit 12 <-> FB Inputs Channel 2/Status/Diag
//     Enc/Inputs/In/nState1 @bit 1 <-> FB Inputs Channel 2/Status/Error
//     Enc/Inputs/In/nState1 @bit 14 <-> FB Inputs Channel 2/Status/Input cycle counter
//     Enc/Inputs/In/nState1 @bit 2 <-> FB Inputs Channel 2/Status/Ready
//     Enc/Inputs/In/nState1 @bit 13 <-> FB Inputs Channel 2/Status/TxPDO State
//     Enc/Inputs/In/nState1 <-> FB Inputs Channel 2/Status/Warning
//   Axes/M5K4 Y <-> Device 1 (EtherCAT)/Term 1 (EK1200)/Term 39 (EK1122)/Term 94 (EK1100)/EL7041-0052_M5K4Y
//     Drive/Inputs/In/nState1 @bit 3 <-> STM Status/Status/Error
//     Drive/Inputs/In/nState1 @bit 5 <-> STM Status/Status/Moving negative
//     Drive/Inputs/In/nState1 @bit 4 <-> STM Status/Status/Moving positive
//     Drive/Inputs/In/nState1 @bit 1 <-> STM Status/Status/Ready
//     Drive/Inputs/In/nState1 <-> STM Status/Status/Ready to enable
//     Drive/Inputs/In/nState1 @bit 6 <-> STM Status/Status/Torque reduced
//     Drive/Inputs/In/nState1 @bit 2 <-> STM Status/Status/Warning
//     Drive/Inputs/In/nState2 @bit 3 <-> STM Status/Status/Digital input 1
//     Drive/Inputs/In/nState2 @bit 4 <-> STM Status/Status/Digital input 2
//     Drive/Inputs/In/nState2 @bit 5 <-> STM Status/Status/Sync error
//     Drive/Inputs/In/nState2 @bit 7 <-> STM Status/Status/TxPDO Toggle
//     Drive/Inputs/In/nState4 @bit 1 <-> WcState/InputToggle
//     Drive/Inputs/In/nState4 <-> WcState/WcState
//     Drive/Outputs/Out/nCtrl1 <-> STM Control/Control/Enable
//     Drive/Outputs/Out/nCtrl1 @bit 2 <-> STM Control/Control/Reduce torque
//     Drive/Outputs/Out/nCtrl1 @bit 1 <-> STM Control/Control/Reset
//     Drive/Outputs/Out/nDataOut2[0] <-> STM Velocity/Velocity
//   Axes/M5K4 Z <-> Device 1 (EtherCAT)/Term 1 (EK1200)/Term 39 (EK1122)/Term 94 (EK1100)/EL5042_M5K4Z_M5K4rY
//     Enc/Inputs/In/nComState @bit 1 <-> WcState/InputToggle
//     Enc/Inputs/In/nComState <-> WcState/WcState
//     Enc/Inputs/In/nDataIn1 <-> FB Inputs Channel 1/Position
//     Enc/Inputs/In/nState1 @bit 12 <-> FB Inputs Channel 1/Status/Diag
//     Enc/Inputs/In/nState1 @bit 1 <-> FB Inputs Channel 1/Status/Error
//     Enc/Inputs/In/nState1 @bit 14 <-> FB Inputs Channel 1/Status/Input cycle counter
//     Enc/Inputs/In/nState1 @bit 2 <-> FB Inputs Channel 1/Status/Ready
//     Enc/Inputs/In/nState1 @bit 13 <-> FB Inputs Channel 1/Status/TxPDO State
//     Enc/Inputs/In/nState1 <-> FB Inputs Channel 1/Status/Warning
//   Axes/M5K4 Z <-> Device 1 (EtherCAT)/Term 1 (EK1200)/Term 39 (EK1122)/Term 94 (EK1100)/EL7041-0052_M5K4Z
//     Drive/Inputs/In/nState1 @bit 3 <-> STM Status/Status/Error
//     Drive/Inputs/In/nState1 @bit 5 <-> STM Status/Status/Moving negative
//     Drive/Inputs/In/nState1 @bit 4 <-> STM Status/Status/Moving positive
//     Drive/Inputs/In/nState1 @bit 1 <-> STM Status/Status/Ready
//     Drive/Inputs/In/nState1 <-> STM Status/Status/Ready to enable
//     Drive/Inputs/In/nState1 @bit 6 <-> STM Status/Status/Torque reduced
//     Drive/Inputs/In/nState1 @bit 2 <-> STM Status/Status/Warning
//     Drive/Inputs/In/nState2 @bit 3 <-> STM Status/Status/Digital input 1
//     Drive/Inputs/In/nState2 @bit 4 <-> STM Status/Status/Digital input 2
//     Drive/Inputs/In/nState2 @bit 5 <-> STM Status/Status/Sync error
//     Drive/Inputs/In/nState2 @bit 7 <-> STM Status/Status/TxPDO Toggle
//     Drive/Inputs/In/nState4 @bit 1 <-> WcState/InputToggle
//     Drive/Inputs/In/nState4 <-> WcState/WcState
//     Drive/Outputs/Out/nCtrl1 <-> STM Control/Control/Enable
//     Drive/Outputs/Out/nCtrl1 @bit 2 <-> STM Control/Control/Reduce torque
//     Drive/Outputs/Out/nCtrl1 @bit 1 <-> STM Control/Control/Reset
//     Drive/Outputs/Out/nDataOut2[0] <-> STM Velocity/Velocity
//   Axes/M5K4 rY <-> Device 1 (EtherCAT)/Term 1 (EK1200)/Term 39 (EK1122)/Term 94 (EK1100)/EL5042_M5K4Z_M5K4rY
//     Enc/Inputs/In/nComState @bit 1 <-> WcState/InputToggle
//     Enc/Inputs/In/nComState <-> WcState/WcState
//     Enc/Inputs/In/nDataIn1 <-> FB Inputs Channel 2/Position
//     Enc/Inputs/In/nState1 @bit 12 <-> FB Inputs Channel 2/Status/Diag
//     Enc/Inputs/In/nState1 @bit 1 <-> FB Inputs Channel 2/Status/Error
//     Enc/Inputs/In/nState1 @bit 14 <-> FB Inputs Channel 2/Status/Input cycle counter
//     Enc/Inputs/In/nState1 @bit 2 <-> FB Inputs Channel 2/Status/Ready
//     Enc/Inputs/In/nState1 @bit 13 <-> FB Inputs Channel 2/Status/TxPDO State
//     Enc/Inputs/In/nState1 <-> FB Inputs Channel 2/Status/Warning
//   Axes/M5K4 rY <-> Device 1 (EtherCAT)/Term 1 (EK1200)/Term 39 (EK1122)/Term 94 (EK1100)/EL7041-0052_M5K4rY
//     Drive/Inputs/In/nState1 @bit 3 <-> STM Status/Status/Error
//     Drive/Inputs/In/nState1 @bit 5 <-> STM Status/Status/Moving negative
//     Drive/Inputs/In/nState1 @bit 4 <-> STM Status/Status/Moving positive
//     Drive/Inputs/In/nState1 @bit 1 <-> STM Status/Status/Ready
//     Drive/Inputs/In/nState1 <-> STM Status/Status/Ready to enable
//     Drive/Inputs/In/nState1 @bit 6 <-> STM Status/Status/Torque reduced
//     Drive/Inputs/In/nState1 @bit 2 <-> STM Status/Status/Warning
//     Drive/Inputs/In/nState2 @bit 3 <-> STM Status/Status/Digital input 1
//     Drive/Inputs/In/nState2 @bit 4 <-> STM Status/Status/Digital input 2
//     Drive/Inputs/In/nState2 @bit 5 <-> STM Status/Status/Sync error
//     Drive/Inputs/In/nState2 @bit 7 <-> STM Status/Status/TxPDO Toggle
//     Drive/Inputs/In/nState4 @bit 1 <-> WcState/InputToggle
//     Drive/Inputs/In/nState4 <-> WcState/WcState
//     Drive/Outputs/Out/nCtrl1 <-> STM Control/Control/Enable
//     Drive/Outputs/Out/nCtrl1 @bit 2 <-> STM Control/Control/Reduce torque
//     Drive/Outputs/Out/nCtrl1 @bit 1 <-> STM Control/Control/Reset
//     Drive/Outputs/Out/nDataOut2[0] <-> STM Velocity/Velocity
//   (this object) <-> Device 1 (EtherCAT)/Term 1 (EK1200)/Term 5 (EK1122)/Term 6 (EK1100)/EL5042_M1K4_Xupdwn
//     Enc/Inputs/In/nComState @bit 1 <-> WcState/InputToggle
//     Enc/Inputs/In/nComState <-> WcState/WcState
//     Enc/Inputs/In/nDataIn1 <-> FB Inputs Channel 1/Position
//     Enc/Inputs/In/nDataIn1 <-> FB Inputs Channel 2/Position
//     Enc/Inputs/In/nState1 @bit 12 <-> FB Inputs Channel 1/Status/Diag
//     Enc/Inputs/In/nState1 @bit 12 <-> FB Inputs Channel 2/Status/Diag
//     Enc/Inputs/In/nState1 @bit 1 <-> FB Inputs Channel 1/Status/Error
//     Enc/Inputs/In/nState1 @bit 1 <-> FB Inputs Channel 2/Status/Error
//     Enc/Inputs/In/nState1 @bit 14 <-> FB Inputs Channel 1/Status/Input cycle counter
//     Enc/Inputs/In/nState1 @bit 14 <-> FB Inputs Channel 2/Status/Input cycle counter
//     Enc/Inputs/In/nState1 @bit 2 <-> FB Inputs Channel 1/Status/Ready
//     Enc/Inputs/In/nState1 @bit 2 <-> FB Inputs Channel 2/Status/Ready
//     Enc/Inputs/In/nState1 @bit 13 <-> FB Inputs Channel 1/Status/TxPDO State
//     Enc/Inputs/In/nState1 @bit 13 <-> FB Inputs Channel 2/Status/TxPDO State
//     Enc/Inputs/In/nState1 <-> FB Inputs Channel 1/Status/Warning
//     Enc/Inputs/In/nState1 <-> FB Inputs Channel 2/Status/Warning
//   (this object) <-> Device 1 (EtherCAT)/Term 1 (EK1200)/Term 5 (EK1122)/Term 6 (EK1100)/EL7041-1000_M1K4_Xup
//     Drive/Inputs/In/nState1 @bit 3 <-> STM Status/Status/Error
//     Drive/Inputs/In/nState1 @bit 5 <-> STM Status/Status/Moving negative
//     Drive/Inputs/In/nState1 @bit 4 <-> STM Status/Status/Moving positive
//     Drive/Inputs/In/nState1 @bit 1 <-> STM Status/Status/Ready
//     Drive/Inputs/In/nState1 <-> STM Status/Status/Ready to enable
//     Drive/Inputs/In/nState1 @bit 6 <-> STM Status/Status/Torque reduced
//     Drive/Inputs/In/nState1 @bit 2 <-> STM Status/Status/Warning
//     Drive/Inputs/In/nState2 @bit 3 <-> STM Status/Status/Digital input 1
//     Drive/Inputs/In/nState2 @bit 4 <-> STM Status/Status/Digital input 2
//     Drive/Inputs/In/nState2 @bit 5 <-> STM Status/Status/Sync error
//     Drive/Inputs/In/nState2 @bit 7 <-> STM Status/Status/TxPDO Toggle
//     Drive/Inputs/In/nState4 @bit 1 <-> WcState/InputToggle
//     Drive/Inputs/In/nState4 <-> WcState/WcState
//     Drive/Outputs/Out/nCtrl1 <-> STM Control/Control/Enable
//     Drive/Outputs/Out/nCtrl1 @bit 2 <-> STM Control/Control/Reduce torque
//     Drive/Outputs/Out/nCtrl1 @bit 1 <-> STM Control/Control/Reset
//     Drive/Outputs/Out/nDataOut2[0] <-> STM Velocity/Velocity
//   (this object) <-> Device 1 (EtherCAT)/Term 1 (EK1200)/Term 5 (EK1122)/Term 6 (EK1100)/EL7041-1000_M1K4_Xdwn
//     Drive/Inputs/In/nState1 @bit 3 <-> STM Status/Status/Error
//     Drive/Inputs/In/nState1 @bit 5 <-> STM Status/Status/Moving negative
//     Drive/Inputs/In/nState1 @bit 4 <-> STM Status/Status/Moving positive
//     Drive/Inputs/In/nState1 @bit 1 <-> STM Status/Status/Ready
//     Drive/Inputs/In/nState1 <-> STM Status/Status/Ready to enable
//     Drive/Inputs/In/nState1 @bit 6 <-> STM Status/Status/Torque reduced
//     Drive/Inputs/In/nState1 @bit 2 <-> STM Status/Status/Warning
//     Drive/Inputs/In/nState2 @bit 3 <-> STM Status/Status/Digital input 1
//     Drive/Inputs/In/nState2 @bit 4 <-> STM Status/Status/Digital input 2
//     Drive/Inputs/In/nState2 @bit 5 <-> STM Status/Status/Sync error
//     Drive/Inputs/In/nState2 @bit 7 <-> STM Status/Status/TxPDO Toggle
//     Drive/Inputs/In/nState4 @bit 1 <-> WcState/InputToggle
//     Drive/Inputs/In/nState4 <-> WcState/WcState
//     Drive/Outputs/Out/nCtrl1 <-> STM Control/Control/Enable
//     Drive/Outputs/Out/nCtrl1 @bit 2 <-> STM Control/Control/Reduce torque
//     Drive/Outputs/Out/nCtrl1 @bit 1 <-> STM Control/Control/Reset
//     Drive/Outputs/Out/nDataOut2[0] <-> STM Velocity/Velocity
//   (this object) <-> Device 1 (EtherCAT)/Term 1 (EK1200)/Term 5 (EK1122)/Term 6 (EK1100)/EL5042_M1K4_PitchBender
//     Enc/Inputs/In/nComState @bit 1 <-> WcState/InputToggle
//     Enc/Inputs/In/nComState <-> WcState/WcState
//     Enc/Inputs/In/nDataIn1 <-> FB Inputs Channel 1/Position
//     Enc/Inputs/In/nDataIn1 <-> FB Inputs Channel 2/Position
//     Enc/Inputs/In/nState1 @bit 12 <-> FB Inputs Channel 1/Status/Diag
//     Enc/Inputs/In/nState1 @bit 12 <-> FB Inputs Channel 2/Status/Diag
//     Enc/Inputs/In/nState1 @bit 1 <-> FB Inputs Channel 1/Status/Error
//     Enc/Inputs/In/nState1 @bit 1 <-> FB Inputs Channel 2/Status/Error
//     Enc/Inputs/In/nState1 @bit 14 <-> FB Inputs Channel 1/Status/Input cycle counter
//     Enc/Inputs/In/nState1 @bit 14 <-> FB Inputs Channel 2/Status/Input cycle counter
//     Enc/Inputs/In/nState1 @bit 2 <-> FB Inputs Channel 1/Status/Ready
//     Enc/Inputs/In/nState1 @bit 2 <-> FB Inputs Channel 2/Status/Ready
//     Enc/Inputs/In/nState1 @bit 13 <-> FB Inputs Channel 1/Status/TxPDO State
//     Enc/Inputs/In/nState1 @bit 13 <-> FB Inputs Channel 2/Status/TxPDO State
//     Enc/Inputs/In/nState1 <-> FB Inputs Channel 1/Status/Warning
//     Enc/Inputs/In/nState1 <-> FB Inputs Channel 2/Status/Warning
//   (this object) <-> Device 1 (EtherCAT)/Term 1 (EK1200)/Term 5 (EK1122)/Term 6 (EK1100)/EL7041-1000_M1K4_PitchCoarse
//     Drive/Inputs/In/nState1 @bit 3 <-> STM Status/Status/Error
//     Drive/Inputs/In/nState1 @bit 5 <-> STM Status/Status/Moving negative
//     Drive/Inputs/In/nState1 @bit 4 <-> STM Status/Status/Moving positive
//     Drive/Inputs/In/nState1 @bit 1 <-> STM Status/Status/Ready
//     Drive/Inputs/In/nState1 <-> STM Status/Status/Ready to enable
//     Drive/Inputs/In/nState1 @bit 6 <-> STM Status/Status/Torque reduced
//     Drive/Inputs/In/nState1 @bit 2 <-> STM Status/Status/Warning
//     Drive/Inputs/In/nState2 @bit 3 <-> STM Status/Status/Digital input 1
//     Drive/Inputs/In/nState2 @bit 4 <-> STM Status/Status/Digital input 2
//     Drive/Inputs/In/nState2 @bit 5 <-> STM Status/Status/Sync error
//     Drive/Inputs/In/nState2 @bit 7 <-> STM Status/Status/TxPDO Toggle
//     Drive/Inputs/In/nState4 @bit 1 <-> WcState/InputToggle
//     Drive/Inputs/In/nState4 <-> WcState/WcState
//     Drive/Outputs/Out/nCtrl1 <-> STM Control/Control/Enable
//     Drive/Outputs/Out/nCtrl1 @bit 2 <-> STM Control/Control/Reduce torque
//     Drive/Outputs/Out/nCtrl1 @bit 1 <-> STM Control/Control/Reset
//     Drive/Outputs/Out/nDataOut2[0] <-> STM Velocity/Velocity
//   (this object) <-> Device 1 (EtherCAT)/Term 1 (EK1200)/Term 5 (EK1122)/Term 20 (EK1100)/EL5042_M2K4X_M2K4Y
//     Enc/Inputs/In/nComState @bit 1 <-> WcState/InputToggle
//     Enc/Inputs/In/nComState <-> WcState/WcState
//     Enc/Inputs/In/nDataIn1 <-> FB Inputs Channel 1/Position
//     Enc/Inputs/In/nDataIn1 <-> FB Inputs Channel 2/Position
//     Enc/Inputs/In/nState1 @bit 12 <-> FB Inputs Channel 1/Status/Diag
//     Enc/Inputs/In/nState1 @bit 12 <-> FB Inputs Channel 2/Status/Diag
//     Enc/Inputs/In/nState1 @bit 1 <-> FB Inputs Channel 1/Status/Error
//     Enc/Inputs/In/nState1 @bit 1 <-> FB Inputs Channel 2/Status/Error
//     Enc/Inputs/In/nState1 @bit 14 <-> FB Inputs Channel 1/Status/Input cycle counter
//     Enc/Inputs/In/nState1 @bit 14 <-> FB Inputs Channel 2/Status/Input cycle counter
//     Enc/Inputs/In/nState1 @bit 2 <-> FB Inputs Channel 1/Status/Ready
//     Enc/Inputs/In/nState1 @bit 2 <-> FB Inputs Channel 2/Status/Ready
//     Enc/Inputs/In/nState1 @bit 13 <-> FB Inputs Channel 1/Status/TxPDO State
//     Enc/Inputs/In/nState1 @bit 13 <-> FB Inputs Channel 2/Status/TxPDO State
//     Enc/Inputs/In/nState1 <-> FB Inputs Channel 1/Status/Warning
//     Enc/Inputs/In/nState1 <-> FB Inputs Channel 2/Status/Warning
//   (this object) <-> Device 1 (EtherCAT)/Term 1 (EK1200)/Term 5 (EK1122)/Term 20 (EK1100)/EL7041-0052_M2K4X
//     Drive/Inputs/In/nState1 @bit 3 <-> STM Status/Status/Error
//     Drive/Inputs/In/nState1 @bit 5 <-> STM Status/Status/Moving negative
//     Drive/Inputs/In/nState1 @bit 4 <-> STM Status/Status/Moving positive
//     Drive/Inputs/In/nState1 @bit 1 <-> STM Status/Status/Ready
//     Drive/Inputs/In/nState1 <-> STM Status/Status/Ready to enable
//     Drive/Inputs/In/nState1 @bit 6 <-> STM Status/Status/Torque reduced
//     Drive/Inputs/In/nState1 @bit 2 <-> STM Status/Status/Warning
//     Drive/Inputs/In/nState2 @bit 3 <-> STM Status/Status/Digital input 1
//     Drive/Inputs/In/nState2 @bit 4 <-> STM Status/Status/Digital input 2
//     Drive/Inputs/In/nState2 @bit 5 <-> STM Status/Status/Sync error
//     Drive/Inputs/In/nState2 @bit 7 <-> STM Status/Status/TxPDO Toggle
//     Drive/Inputs/In/nState4 @bit 1 <-> WcState/InputToggle
//     Drive/Inputs/In/nState4 <-> WcState/WcState
//     Drive/Outputs/Out/nCtrl1 <-> STM Control/Control/Enable
//     Drive/Outputs/Out/nCtrl1 @bit 2 <-> STM Control/Control/Reduce torque
//     Drive/Outputs/Out/nCtrl1 @bit 1 <-> STM Control/Control/Reset
//     Drive/Outputs/Out/nDataOut2[0] <-> STM Velocity/Velocity
//   (this object) <-> Device 1 (EtherCAT)/Term 1 (EK1200)/Term 5 (EK1122)/Term 20 (EK1100)/EL7041-0052_M2K4Y
//     Drive/Inputs/In/nState1 @bit 3 <-> STM Status/Status/Error
//     Drive/Inputs/In/nState1 @bit 5 <-> STM Status/Status/Moving negative
//     Drive/Inputs/In/nState1 @bit 4 <-> STM Status/Status/Moving positive
//     Drive/Inputs/In/nState1 @bit 1 <-> STM Status/Status/Ready
//     Drive/Inputs/In/nState1 <-> STM Status/Status/Ready to enable
//     Drive/Inputs/In/nState1 @bit 6 <-> STM Status/Status/Torque reduced
//     Drive/Inputs/In/nState1 @bit 2 <-> STM Status/Status/Warning
//     Drive/Inputs/In/nState2 @bit 3 <-> STM Status/Status/Digital input 1
//     Drive/Inputs/In/nState2 @bit 4 <-> STM Status/Status/Digital input 2
//     Drive/Inputs/In/nState2 @bit 5 <-> STM Status/Status/Sync error
//     Drive/Inputs/In/nState2 @bit 7 <-> STM Status/Status/TxPDO Toggle
//     Drive/Inputs/In/nState4 @bit 1 <-> WcState/InputToggle
//     Drive/Inputs/In/nState4 <-> WcState/WcState
//     Drive/Outputs/Out/nCtrl1 <-> STM Control/Control/Enable
//     Drive/Outputs/Out/nCtrl1 @bit 2 <-> STM Control/Control/Reduce torque
//     Drive/Outputs/Out/nCtrl1 @bit 1 <-> STM Control/Control/Reset
//     Drive/Outputs/Out/nDataOut2[0] <-> STM Velocity/Velocity
//   (this object) <-> Device 1 (EtherCAT)/Term 1 (EK1200)/Term 5 (EK1122)/Term 20 (EK1100)/EL5042_M2K4rY_M3K4X
//     Enc/Inputs/In/nComState @bit 1 <-> WcState/InputToggle
//     Enc/Inputs/In/nComState <-> WcState/WcState
//     Enc/Inputs/In/nDataIn1 <-> FB Inputs Channel 1/Position
//     Enc/Inputs/In/nDataIn1 <-> FB Inputs Channel 2/Position
//     Enc/Inputs/In/nState1 @bit 12 <-> FB Inputs Channel 1/Status/Diag
//     Enc/Inputs/In/nState1 @bit 12 <-> FB Inputs Channel 2/Status/Diag
//     Enc/Inputs/In/nState1 @bit 1 <-> FB Inputs Channel 1/Status/Error
//     Enc/Inputs/In/nState1 @bit 1 <-> FB Inputs Channel 2/Status/Error
//     Enc/Inputs/In/nState1 @bit 14 <-> FB Inputs Channel 1/Status/Input cycle counter
//     Enc/Inputs/In/nState1 @bit 14 <-> FB Inputs Channel 2/Status/Input cycle counter
//     Enc/Inputs/In/nState1 @bit 2 <-> FB Inputs Channel 1/Status/Ready
//     Enc/Inputs/In/nState1 @bit 2 <-> FB Inputs Channel 2/Status/Ready
//     Enc/Inputs/In/nState1 @bit 13 <-> FB Inputs Channel 1/Status/TxPDO State
//     Enc/Inputs/In/nState1 @bit 13 <-> FB Inputs Channel 2/Status/TxPDO State
//     Enc/Inputs/In/nState1 <-> FB Inputs Channel 1/Status/Warning
//     Enc/Inputs/In/nState1 <-> FB Inputs Channel 2/Status/Warning
//   (this object) <-> Device 1 (EtherCAT)/Term 1 (EK1200)/Term 5 (EK1122)/Term 20 (EK1100)/EL7041-0052_M2K4rY
//     Drive/Inputs/In/nState1 @bit 3 <-> STM Status/Status/Error
//     Drive/Inputs/In/nState1 @bit 5 <-> STM Status/Status/Moving negative
//     Drive/Inputs/In/nState1 @bit 4 <-> STM Status/Status/Moving positive
//     Drive/Inputs/In/nState1 @bit 1 <-> STM Status/Status/Ready
//     Drive/Inputs/In/nState1 <-> STM Status/Status/Ready to enable
//     Drive/Inputs/In/nState1 @bit 6 <-> STM Status/Status/Torque reduced
//     Drive/Inputs/In/nState1 @bit 2 <-> STM Status/Status/Warning
//     Drive/Inputs/In/nState2 @bit 3 <-> STM Status/Status/Digital input 1
//     Drive/Inputs/In/nState2 @bit 4 <-> STM Status/Status/Digital input 2
//     Drive/Inputs/In/nState2 @bit 5 <-> STM Status/Status/Sync error
//     Drive/Inputs/In/nState2 @bit 7 <-> STM Status/Status/TxPDO Toggle
//     Drive/Inputs/In/nState4 @bit 1 <-> WcState/InputToggle
//     Drive/Inputs/In/nState4 <-> WcState/WcState
//     Drive/Outputs/Out/nCtrl1 <-> STM Control/Control/Enable
//     Drive/Outputs/Out/nCtrl1 @bit 2 <-> STM Control/Control/Reduce torque
//     Drive/Outputs/Out/nCtrl1 @bit 1 <-> STM Control/Control/Reset
//     Drive/Outputs/Out/nDataOut2[0] <-> STM Velocity/Velocity
//   (this object) <-> Device 1 (EtherCAT)/Term 1 (EK1200)/Term 5 (EK1122)/Term 20 (EK1100)/EL5042_M2K4_BEND_USDS
//     Enc/Inputs/In/nComState @bit 1 <-> WcState/InputToggle
//     Enc/Inputs/In/nComState <-> WcState/WcState
//     Enc/Inputs/In/nDataIn1 <-> FB Inputs Channel 1/Position
//     Enc/Inputs/In/nDataIn1 <-> FB Inputs Channel 2/Position
//     Enc/Inputs/In/nState1 @bit 12 <-> FB Inputs Channel 1/Status/Diag
//     Enc/Inputs/In/nState1 @bit 12 <-> FB Inputs Channel 2/Status/Diag
//     Enc/Inputs/In/nState1 @bit 1 <-> FB Inputs Channel 1/Status/Error
//     Enc/Inputs/In/nState1 @bit 1 <-> FB Inputs Channel 2/Status/Error
//     Enc/Inputs/In/nState1 @bit 14 <-> FB Inputs Channel 1/Status/Input cycle counter
//     Enc/Inputs/In/nState1 @bit 14 <-> FB Inputs Channel 2/Status/Input cycle counter
//     Enc/Inputs/In/nState1 @bit 2 <-> FB Inputs Channel 1/Status/Ready
//     Enc/Inputs/In/nState1 @bit 2 <-> FB Inputs Channel 2/Status/Ready
//     Enc/Inputs/In/nState1 @bit 13 <-> FB Inputs Channel 1/Status/TxPDO State
//     Enc/Inputs/In/nState1 @bit 13 <-> FB Inputs Channel 2/Status/TxPDO State
//     Enc/Inputs/In/nState1 <-> FB Inputs Channel 1/Status/Warning
//     Enc/Inputs/In/nState1 <-> FB Inputs Channel 2/Status/Warning
//   (this object) <-> Device 1 (EtherCAT)/Term 1 (EK1200)/Term 5 (EK1122)/Term 20 (EK1100)/EL7041_M2K4_BEND_US
//     Drive/Inputs/In/nState1 @bit 3 <-> STM Status/Status/Error
//     Drive/Inputs/In/nState1 @bit 5 <-> STM Status/Status/Moving negative
//     Drive/Inputs/In/nState1 @bit 4 <-> STM Status/Status/Moving positive
//     Drive/Inputs/In/nState1 @bit 1 <-> STM Status/Status/Ready
//     Drive/Inputs/In/nState1 <-> STM Status/Status/Ready to enable
//     Drive/Inputs/In/nState1 @bit 6 <-> STM Status/Status/Torque reduced
//     Drive/Inputs/In/nState1 @bit 2 <-> STM Status/Status/Warning
//     Drive/Inputs/In/nState2 @bit 3 <-> STM Status/Status/Digital input 1
//     Drive/Inputs/In/nState2 @bit 4 <-> STM Status/Status/Digital input 2
//     Drive/Inputs/In/nState2 @bit 5 <-> STM Status/Status/Sync error
//     Drive/Inputs/In/nState2 @bit 7 <-> STM Status/Status/TxPDO Toggle
//     Drive/Inputs/In/nState4 @bit 1 <-> WcState/InputToggle
//     Drive/Inputs/In/nState4 <-> WcState/WcState
//     Drive/Outputs/Out/nCtrl1 <-> STM Control/Control/Enable
//     Drive/Outputs/Out/nCtrl1 @bit 2 <-> STM Control/Control/Reduce torque
//     Drive/Outputs/Out/nCtrl1 @bit 1 <-> STM Control/Control/Reset
//     Drive/Outputs/Out/nDataOut2[0] <-> STM Velocity/Velocity
//   (this object) <-> Device 1 (EtherCAT)/Term 1 (EK1200)/Term 5 (EK1122)/Term 20 (EK1100)/EL7041_M2K4_BEND_DS
//     Drive/Inputs/In/nState1 @bit 3 <-> STM Status/Status/Error
//     Drive/Inputs/In/nState1 @bit 5 <-> STM Status/Status/Moving negative
//     Drive/Inputs/In/nState1 @bit 4 <-> STM Status/Status/Moving positive
//     Drive/Inputs/In/nState1 @bit 1 <-> STM Status/Status/Ready
//     Drive/Inputs/In/nState1 <-> STM Status/Status/Ready to enable
//     Drive/Inputs/In/nState1 @bit 6 <-> STM Status/Status/Torque reduced
//     Drive/Inputs/In/nState1 @bit 2 <-> STM Status/Status/Warning
//     Drive/Inputs/In/nState2 @bit 3 <-> STM Status/Status/Digital input 1
//     Drive/Inputs/In/nState2 @bit 4 <-> STM Status/Status/Digital input 2
//     Drive/Inputs/In/nState2 @bit 5 <-> STM Status/Status/Sync error
//     Drive/Inputs/In/nState2 @bit 7 <-> STM Status/Status/TxPDO Toggle
//     Drive/Inputs/In/nState4 @bit 1 <-> WcState/InputToggle
//     Drive/Inputs/In/nState4 <-> WcState/WcState
//     Drive/Outputs/Out/nCtrl1 <-> STM Control/Control/Enable
//     Drive/Outputs/Out/nCtrl1 @bit 2 <-> STM Control/Control/Reduce torque
//     Drive/Outputs/Out/nCtrl1 @bit 1 <-> STM Control/Control/Reset
//     Drive/Outputs/Out/nDataOut2[0] <-> STM Velocity/Velocity
//   (this object) <-> Device 1 (EtherCAT)/Term 1 (EK1200)/Term 5 (EK1122)/Term 20 (EK1100)/EL7041-0052_M3K4X
//     Drive/Inputs/In/nState1 @bit 3 <-> STM Status/Status/Error
//     Drive/Inputs/In/nState1 @bit 5 <-> STM Status/Status/Moving negative
//     Drive/Inputs/In/nState1 @bit 4 <-> STM Status/Status/Moving positive
//     Drive/Inputs/In/nState1 @bit 1 <-> STM Status/Status/Ready
//     Drive/Inputs/In/nState1 <-> STM Status/Status/Ready to enable
//     Drive/Inputs/In/nState1 @bit 6 <-> STM Status/Status/Torque reduced
//     Drive/Inputs/In/nState1 @bit 2 <-> STM Status/Status/Warning
//     Drive/Inputs/In/nState2 @bit 3 <-> STM Status/Status/Digital input 1
//     Drive/Inputs/In/nState2 @bit 4 <-> STM Status/Status/Digital input 2
//     Drive/Inputs/In/nState2 @bit 5 <-> STM Status/Status/Sync error
//     Drive/Inputs/In/nState2 @bit 7 <-> STM Status/Status/TxPDO Toggle
//     Drive/Inputs/In/nState4 @bit 1 <-> WcState/InputToggle
//     Drive/Inputs/In/nState4 <-> WcState/WcState
//     Drive/Outputs/Out/nCtrl1 <-> STM Control/Control/Enable
//     Drive/Outputs/Out/nCtrl1 @bit 2 <-> STM Control/Control/Reduce torque
//     Drive/Outputs/Out/nCtrl1 @bit 1 <-> STM Control/Control/Reset
//     Drive/Outputs/Out/nDataOut2[0] <-> STM Velocity/Velocity
//   (this object) <-> Device 1 (EtherCAT)/Term 1 (EK1200)/Term 5 (EK1122)/Term 20 (EK1100)/EL5042_M3K4Y_M3K4rX
//     Enc/Inputs/In/nComState @bit 1 <-> WcState/InputToggle
//     Enc/Inputs/In/nComState <-> WcState/WcState
//     Enc/Inputs/In/nDataIn1 <-> FB Inputs Channel 1/Position
//     Enc/Inputs/In/nDataIn1 <-> FB Inputs Channel 2/Position
//     Enc/Inputs/In/nState1 @bit 12 <-> FB Inputs Channel 1/Status/Diag
//     Enc/Inputs/In/nState1 @bit 12 <-> FB Inputs Channel 2/Status/Diag
//     Enc/Inputs/In/nState1 @bit 1 <-> FB Inputs Channel 1/Status/Error
//     Enc/Inputs/In/nState1 @bit 1 <-> FB Inputs Channel 2/Status/Error
//     Enc/Inputs/In/nState1 @bit 14 <-> FB Inputs Channel 1/Status/Input cycle counter
//     Enc/Inputs/In/nState1 @bit 14 <-> FB Inputs Channel 2/Status/Input cycle counter
//     Enc/Inputs/In/nState1 @bit 2 <-> FB Inputs Channel 1/Status/Ready
//     Enc/Inputs/In/nState1 @bit 2 <-> FB Inputs Channel 2/Status/Ready
//     Enc/Inputs/In/nState1 @bit 13 <-> FB Inputs Channel 1/Status/TxPDO State
//     Enc/Inputs/In/nState1 @bit 13 <-> FB Inputs Channel 2/Status/TxPDO State
//     Enc/Inputs/In/nState1 <-> FB Inputs Channel 1/Status/Warning
//     Enc/Inputs/In/nState1 <-> FB Inputs Channel 2/Status/Warning
//   (this object) <-> Device 1 (EtherCAT)/Term 1 (EK1200)/Term 5 (EK1122)/Term 20 (EK1100)/EL7041-0052_M3K4Y
//     Drive/Inputs/In/nState1 @bit 3 <-> STM Status/Status/Error
//     Drive/Inputs/In/nState1 @bit 5 <-> STM Status/Status/Moving negative
//     Drive/Inputs/In/nState1 @bit 4 <-> STM Status/Status/Moving positive
//     Drive/Inputs/In/nState1 @bit 1 <-> STM Status/Status/Ready
//     Drive/Inputs/In/nState1 <-> STM Status/Status/Ready to enable
//     Drive/Inputs/In/nState1 @bit 6 <-> STM Status/Status/Torque reduced
//     Drive/Inputs/In/nState1 @bit 2 <-> STM Status/Status/Warning
//     Drive/Inputs/In/nState2 @bit 3 <-> STM Status/Status/Digital input 1
//     Drive/Inputs/In/nState2 @bit 4 <-> STM Status/Status/Digital input 2
//     Drive/Inputs/In/nState2 @bit 5 <-> STM Status/Status/Sync error
//     Drive/Inputs/In/nState2 @bit 7 <-> STM Status/Status/TxPDO Toggle
//     Drive/Inputs/In/nState4 @bit 1 <-> WcState/InputToggle
//     Drive/Inputs/In/nState4 <-> WcState/WcState
//     Drive/Outputs/Out/nCtrl1 <-> STM Control/Control/Enable
//     Drive/Outputs/Out/nCtrl1 @bit 2 <-> STM Control/Control/Reduce torque
//     Drive/Outputs/Out/nCtrl1 @bit 1 <-> STM Control/Control/Reset
//     Drive/Outputs/Out/nDataOut2[0] <-> STM Velocity/Velocity
//   (this object) <-> Device 1 (EtherCAT)/Term 1 (EK1200)/Term 5 (EK1122)/Term 20 (EK1100)/EL7041-0052_M3K4rX
//     Drive/Inputs/In/nState1 @bit 3 <-> STM Status/Status/Error
//     Drive/Inputs/In/nState1 @bit 5 <-> STM Status/Status/Moving negative
//     Drive/Inputs/In/nState1 @bit 4 <-> STM Status/Status/Moving positive
//     Drive/Inputs/In/nState1 @bit 1 <-> STM Status/Status/Ready
//     Drive/Inputs/In/nState1 <-> STM Status/Status/Ready to enable
//     Drive/Inputs/In/nState1 @bit 6 <-> STM Status/Status/Torque reduced
//     Drive/Inputs/In/nState1 @bit 2 <-> STM Status/Status/Warning
//     Drive/Inputs/In/nState2 @bit 3 <-> STM Status/Status/Digital input 1
//     Drive/Inputs/In/nState2 @bit 4 <-> STM Status/Status/Digital input 2
//     Drive/Inputs/In/nState2 @bit 5 <-> STM Status/Status/Sync error
//     Drive/Inputs/In/nState2 @bit 7 <-> STM Status/Status/TxPDO Toggle
//     Drive/Inputs/In/nState4 @bit 1 <-> WcState/InputToggle
//     Drive/Inputs/In/nState4 <-> WcState/WcState
//     Drive/Outputs/Out/nCtrl1 <-> STM Control/Control/Enable
//     Drive/Outputs/Out/nCtrl1 @bit 2 <-> STM Control/Control/Reduce torque
//     Drive/Outputs/Out/nCtrl1 @bit 1 <-> STM Control/Control/Reset
//     Drive/Outputs/Out/nDataOut2[0] <-> STM Velocity/Velocity
//   (this object) <-> Device 1 (EtherCAT)/Term 1 (EK1200)/Term 5 (EK1122)/Term 20 (EK1100)/EL5042_M3K4_BEND_USDS
//     Enc/Inputs/In/nComState @bit 1 <-> WcState/InputToggle
//     Enc/Inputs/In/nComState <-> WcState/WcState
//     Enc/Inputs/In/nDataIn1 <-> FB Inputs Channel 1/Position
//     Enc/Inputs/In/nDataIn1 <-> FB Inputs Channel 2/Position
//     Enc/Inputs/In/nState1 @bit 12 <-> FB Inputs Channel 1/Status/Diag
//     Enc/Inputs/In/nState1 @bit 12 <-> FB Inputs Channel 2/Status/Diag
//     Enc/Inputs/In/nState1 @bit 1 <-> FB Inputs Channel 1/Status/Error
//     Enc/Inputs/In/nState1 @bit 1 <-> FB Inputs Channel 2/Status/Error
//     Enc/Inputs/In/nState1 @bit 14 <-> FB Inputs Channel 1/Status/Input cycle counter
//     Enc/Inputs/In/nState1 @bit 14 <-> FB Inputs Channel 2/Status/Input cycle counter
//     Enc/Inputs/In/nState1 @bit 2 <-> FB Inputs Channel 1/Status/Ready
//     Enc/Inputs/In/nState1 @bit 2 <-> FB Inputs Channel 2/Status/Ready
//     Enc/Inputs/In/nState1 @bit 13 <-> FB Inputs Channel 1/Status/TxPDO State
//     Enc/Inputs/In/nState1 @bit 13 <-> FB Inputs Channel 2/Status/TxPDO State
//     Enc/Inputs/In/nState1 <-> FB Inputs Channel 1/Status/Warning
//     Enc/Inputs/In/nState1 <-> FB Inputs Channel 2/Status/Warning
//   (this object) <-> Device 1 (EtherCAT)/Term 1 (EK1200)/Term 5 (EK1122)/Term 20 (EK1100)/EL7041_M3K4_BEND_US
//     Drive/Inputs/In/nState1 @bit 3 <-> STM Status/Status/Error
//     Drive/Inputs/In/nState1 @bit 5 <-> STM Status/Status/Moving negative
//     Drive/Inputs/In/nState1 @bit 4 <-> STM Status/Status/Moving positive
//     Drive/Inputs/In/nState1 @bit 1 <-> STM Status/Status/Ready
//     Drive/Inputs/In/nState1 <-> STM Status/Status/Ready to enable
//     Drive/Inputs/In/nState1 @bit 6 <-> STM Status/Status/Torque reduced
//     Drive/Inputs/In/nState1 @bit 2 <-> STM Status/Status/Warning
//     Drive/Inputs/In/nState2 @bit 3 <-> STM Status/Status/Digital input 1
//     Drive/Inputs/In/nState2 @bit 4 <-> STM Status/Status/Digital input 2
//     Drive/Inputs/In/nState2 @bit 5 <-> STM Status/Status/Sync error
//     Drive/Inputs/In/nState2 @bit 7 <-> STM Status/Status/TxPDO Toggle
//     Drive/Inputs/In/nState4 @bit 1 <-> WcState/InputToggle
//     Drive/Inputs/In/nState4 <-> WcState/WcState
//     Drive/Outputs/Out/nCtrl1 <-> STM Control/Control/Enable
//     Drive/Outputs/Out/nCtrl1 @bit 2 <-> STM Control/Control/Reduce torque
//     Drive/Outputs/Out/nCtrl1 @bit 1 <-> STM Control/Control/Reset
//     Drive/Outputs/Out/nDataOut2[0] <-> STM Velocity/Velocity
//   (this object) <-> Device 1 (EtherCAT)/Term 1 (EK1200)/Term 5 (EK1122)/Term 20 (EK1100)/EL7041_M3K4_BEND_DS
//     Drive/Inputs/In/nState1 @bit 3 <-> STM Status/Status/Error
//     Drive/Inputs/In/nState1 @bit 5 <-> STM Status/Status/Moving negative
//     Drive/Inputs/In/nState1 @bit 4 <-> STM Status/Status/Moving positive
//     Drive/Inputs/In/nState1 @bit 1 <-> STM Status/Status/Ready
//     Drive/Inputs/In/nState1 <-> STM Status/Status/Ready to enable
//     Drive/Inputs/In/nState1 @bit 6 <-> STM Status/Status/Torque reduced
//     Drive/Inputs/In/nState1 @bit 2 <-> STM Status/Status/Warning
//     Drive/Inputs/In/nState2 @bit 3 <-> STM Status/Status/Digital input 1
//     Drive/Inputs/In/nState2 @bit 4 <-> STM Status/Status/Digital input 2
//     Drive/Inputs/In/nState2 @bit 5 <-> STM Status/Status/Sync error
//     Drive/Inputs/In/nState2 @bit 7 <-> STM Status/Status/TxPDO Toggle
//     Drive/Inputs/In/nState4 @bit 1 <-> WcState/InputToggle
//     Drive/Inputs/In/nState4 <-> WcState/WcState
//     Drive/Outputs/Out/nCtrl1 <-> STM Control/Control/Enable
//     Drive/Outputs/Out/nCtrl1 @bit 2 <-> STM Control/Control/Reduce torque
//     Drive/Outputs/Out/nCtrl1 @bit 1 <-> STM Control/Control/Reset
//     Drive/Outputs/Out/nDataOut2[0] <-> STM Velocity/Velocity
//   (this object) <-> Device 1 (EtherCAT)/Term 1 (EK1200)/Term 39 (EK1122)/B940-009-R19-DRL-04 (EK1100)/SL2K4-EL7031-E3
//     Drive/Inputs/In/nState1 @bit 3 <-> STM Status/Status/Error
//     Drive/Inputs/In/nState1 @bit 5 <-> STM Status/Status/Moving negative
//     Drive/Inputs/In/nState1 @bit 4 <-> STM Status/Status/Moving positive
//     Drive/Inputs/In/nState1 @bit 1 <-> STM Status/Status/Ready
//     Drive/Inputs/In/nState1 <-> STM Status/Status/Ready to enable
//     Drive/Inputs/In/nState1 @bit 6 <-> STM Status/Status/Torque reduced
//     Drive/Inputs/In/nState1 @bit 2 <-> STM Status/Status/Warning
//     Drive/Inputs/In/nState2 @bit 3 <-> STM Status/Status/Digital input 1
//     Drive/Inputs/In/nState2 @bit 4 <-> STM Status/Status/Digital input 2
//     Drive/Inputs/In/nState2 @bit 5 <-> STM Status/Status/Sync error
//     Drive/Inputs/In/nState2 @bit 7 <-> STM Status/Status/TxPDO Toggle
//     Drive/Inputs/In/nState4 @bit 1 <-> WcState/InputToggle
//     Drive/Inputs/In/nState4 <-> WcState/WcState
//     Drive/Outputs/Out/nCtrl1 <-> STM Control/Control/Enable
//     Drive/Outputs/Out/nCtrl1 @bit 2 <-> STM Control/Control/Reduce torque
//     Drive/Outputs/Out/nCtrl1 @bit 1 <-> STM Control/Control/Reset
//     Drive/Outputs/Out/nDataOut2[0] <-> STM Velocity/Velocity
//     Enc/Inputs/In/nDataIn2[0] <-> ENC Status compact/Latch value
//     Enc/Inputs/In/nState1 @bit 4 <-> ENC Status compact/Status/Counter overflow
//     Enc/Inputs/In/nState1 @bit 3 <-> ENC Status compact/Status/Counter underflow
//     Enc/Inputs/In/nState1 @bit 1 <-> ENC Status compact/Status/Latch extern valid
//     Enc/Inputs/In/nState1 @bit 2 <-> ENC Status compact/Status/Set counter done
//     Enc/Inputs/In/nState2 @bit 4 <-> ENC Status compact/Status/Status of extern latch
//     Enc/Inputs/In/nState2 @bit 5 <-> ENC Status compact/Status/Sync error
//     Enc/Inputs/In/nState2 @bit 7 <-> ENC Status compact/Status/TxPDO Toggle
//     Enc/Inputs/In/nState4 @bit 1 <-> WcState/InputToggle
//     Enc/Inputs/In/nState4 <-> WcState/WcState
//     Enc/Outputs/Out/nCtrl1 @bit 3 <-> ENC Control compact/Control/Enable latch extern on negative edge
//     Enc/Outputs/Out/nCtrl1 @bit 1 <-> ENC Control compact/Control/Enable latch extern on positive edge
//     Enc/Outputs/Out/nCtrl1 @bit 2 <-> ENC Control compact/Control/Set counter
//     Enc/Outputs/Out/nDataOut1[0] <-> ENC Control compact/Set counter value
//   (this object) <-> Device 1 (EtherCAT)/Term 1 (EK1200)/Term 39 (EK1122)/B940-009-R19-DRL-04 (EK1100)/SL2K4-EL7031-E4
//     Drive/Inputs/In/nState1 @bit 3 <-> STM Status/Status/Error
//     Drive/Inputs/In/nState1 @bit 5 <-> STM Status/Status/Moving negative
//     Drive/Inputs/In/nState1 @bit 4 <-> STM Status/Status/Moving positive
//     Drive/Inputs/In/nState1 @bit 1 <-> STM Status/Status/Ready
//     Drive/Inputs/In/nState1 <-> STM Status/Status/Ready to enable
//     Drive/Inputs/In/nState1 @bit 6 <-> STM Status/Status/Torque reduced
//     Drive/Inputs/In/nState1 @bit 2 <-> STM Status/Status/Warning
//     Drive/Inputs/In/nState2 @bit 3 <-> STM Status/Status/Digital input 1
//     Drive/Inputs/In/nState2 @bit 4 <-> STM Status/Status/Digital input 2
//     Drive/Inputs/In/nState2 @bit 5 <-> STM Status/Status/Sync error
//     Drive/Inputs/In/nState2 @bit 7 <-> STM Status/Status/TxPDO Toggle
//     Drive/Inputs/In/nState4 @bit 1 <-> WcState/InputToggle
//     Drive/Inputs/In/nState4 <-> WcState/WcState
//     Drive/Outputs/Out/nCtrl1 <-> STM Control/Control/Enable
//     Drive/Outputs/Out/nCtrl1 @bit 2 <-> STM Control/Control/Reduce torque
//     Drive/Outputs/Out/nCtrl1 @bit 1 <-> STM Control/Control/Reset
//     Drive/Outputs/Out/nDataOut2[0] <-> STM Velocity/Velocity
//     Enc/Inputs/In/nDataIn2[0] <-> ENC Status compact/Latch value
//     Enc/Inputs/In/nState1 @bit 4 <-> ENC Status compact/Status/Counter overflow
//     Enc/Inputs/In/nState1 @bit 3 <-> ENC Status compact/Status/Counter underflow
//     Enc/Inputs/In/nState1 @bit 1 <-> ENC Status compact/Status/Latch extern valid
//     Enc/Inputs/In/nState1 @bit 2 <-> ENC Status compact/Status/Set counter done
//     Enc/Inputs/In/nState2 @bit 4 <-> ENC Status compact/Status/Status of extern latch
//     Enc/Inputs/In/nState2 @bit 5 <-> ENC Status compact/Status/Sync error
//     Enc/Inputs/In/nState2 @bit 7 <-> ENC Status compact/Status/TxPDO Toggle
//     Enc/Inputs/In/nState4 @bit 1 <-> WcState/InputToggle
//     Enc/Inputs/In/nState4 <-> WcState/WcState
//     Enc/Outputs/Out/nCtrl1 @bit 3 <-> ENC Control compact/Control/Enable latch extern on negative edge
//     Enc/Outputs/Out/nCtrl1 @bit 1 <-> ENC Control compact/Control/Enable latch extern on positive edge
//     Enc/Outputs/Out/nCtrl1 @bit 2 <-> ENC Control compact/Control/Set counter
//     Enc/Outputs/Out/nDataOut1[0] <-> ENC Control compact/Set counter value
//   (this object) <-> Device 1 (EtherCAT)/Term 1 (EK1200)/Term 39 (EK1122)/B940-009-R19-DRL-04 (EK1100)/SL2K4-EL7031-E5
//     Drive/Inputs/In/nState1 @bit 3 <-> STM Status/Status/Error
//     Drive/Inputs/In/nState1 @bit 5 <-> STM Status/Status/Moving negative
//     Drive/Inputs/In/nState1 @bit 4 <-> STM Status/Status/Moving positive
//     Drive/Inputs/In/nState1 @bit 1 <-> STM Status/Status/Ready
//     Drive/Inputs/In/nState1 <-> STM Status/Status/Ready to enable
//     Drive/Inputs/In/nState1 @bit 6 <-> STM Status/Status/Torque reduced
//     Drive/Inputs/In/nState1 @bit 2 <-> STM Status/Status/Warning
//     Drive/Inputs/In/nState2 @bit 3 <-> STM Status/Status/Digital input 1
//     Drive/Inputs/In/nState2 @bit 4 <-> STM Status/Status/Digital input 2
//     Drive/Inputs/In/nState2 @bit 5 <-> STM Status/Status/Sync error
//     Drive/Inputs/In/nState2 @bit 7 <-> STM Status/Status/TxPDO Toggle
//     Drive/Inputs/In/nState4 @bit 1 <-> WcState/InputToggle
//     Drive/Inputs/In/nState4 <-> WcState/WcState
//     Drive/Outputs/Out/nCtrl1 <-> STM Control/Control/Enable
//     Drive/Outputs/Out/nCtrl1 @bit 2 <-> STM Control/Control/Reduce torque
//     Drive/Outputs/Out/nCtrl1 @bit 1 <-> STM Control/Control/Reset
//     Drive/Outputs/Out/nDataOut2[0] <-> STM Velocity/Velocity
//     Enc/Inputs/In/nDataIn2[0] <-> ENC Status compact/Latch value
//     Enc/Inputs/In/nState1 @bit 4 <-> ENC Status compact/Status/Counter overflow
//     Enc/Inputs/In/nState1 @bit 3 <-> ENC Status compact/Status/Counter underflow
//     Enc/Inputs/In/nState1 @bit 1 <-> ENC Status compact/Status/Latch extern valid
//     Enc/Inputs/In/nState1 @bit 2 <-> ENC Status compact/Status/Set counter done
//     Enc/Inputs/In/nState2 @bit 4 <-> ENC Status compact/Status/Status of extern latch
//     Enc/Inputs/In/nState2 @bit 5 <-> ENC Status compact/Status/Sync error
//     Enc/Inputs/In/nState2 @bit 7 <-> ENC Status compact/Status/TxPDO Toggle
//     Enc/Inputs/In/nState4 @bit 1 <-> WcState/InputToggle
//     Enc/Inputs/In/nState4 <-> WcState/WcState
//     Enc/Outputs/Out/nCtrl1 @bit 3 <-> ENC Control compact/Control/Enable latch extern on negative edge
//     Enc/Outputs/Out/nCtrl1 @bit 1 <-> ENC Control compact/Control/Enable latch extern on positive edge
//     Enc/Outputs/Out/nCtrl1 @bit 2 <-> ENC Control compact/Control/Set counter
//     Enc/Outputs/Out/nDataOut1[0] <-> ENC Control compact/Set counter value
//   (this object) <-> Device 1 (EtherCAT)/Term 1 (EK1200)/Term 39 (EK1122)/B940-009-R19-DRL-04 (EK1100)/SL2K4-EL7031-E6
//     Drive/Inputs/In/nState1 @bit 3 <-> STM Status/Status/Error
//     Drive/Inputs/In/nState1 @bit 5 <-> STM Status/Status/Moving negative
//     Drive/Inputs/In/nState1 @bit 4 <-> STM Status/Status/Moving positive
//     Drive/Inputs/In/nState1 @bit 1 <-> STM Status/Status/Ready
//     Drive/Inputs/In/nState1 <-> STM Status/Status/Ready to enable
//     Drive/Inputs/In/nState1 @bit 6 <-> STM Status/Status/Torque reduced
//     Drive/Inputs/In/nState1 @bit 2 <-> STM Status/Status/Warning
//     Drive/Inputs/In/nState2 @bit 3 <-> STM Status/Status/Digital input 1
//     Drive/Inputs/In/nState2 @bit 4 <-> STM Status/Status/Digital input 2
//     Drive/Inputs/In/nState2 @bit 5 <-> STM Status/Status/Sync error
//     Drive/Inputs/In/nState2 @bit 7 <-> STM Status/Status/TxPDO Toggle
//     Drive/Inputs/In/nState4 @bit 1 <-> WcState/InputToggle
//     Drive/Inputs/In/nState4 <-> WcState/WcState
//     Drive/Outputs/Out/nCtrl1 <-> STM Control/Control/Enable
//     Drive/Outputs/Out/nCtrl1 @bit 2 <-> STM Control/Control/Reduce torque
//     Drive/Outputs/Out/nCtrl1 @bit 1 <-> STM Control/Control/Reset
//     Drive/Outputs/Out/nDataOut2[0] <-> STM Velocity/Velocity
//     Enc/Inputs/In/nDataIn2[0] <-> ENC Status compact/Latch value
//     Enc/Inputs/In/nState1 @bit 4 <-> ENC Status compact/Status/Counter overflow
//     Enc/Inputs/In/nState1 @bit 3 <-> ENC Status compact/Status/Counter underflow
//     Enc/Inputs/In/nState1 @bit 1 <-> ENC Status compact/Status/Latch extern valid
//     Enc/Inputs/In/nState1 @bit 2 <-> ENC Status compact/Status/Set counter done
//     Enc/Inputs/In/nState2 @bit 4 <-> ENC Status compact/Status/Status of extern latch
//     Enc/Inputs/In/nState2 @bit 5 <-> ENC Status compact/Status/Sync error
//     Enc/Inputs/In/nState2 @bit 7 <-> ENC Status compact/Status/TxPDO Toggle
//     Enc/Inputs/In/nState4 @bit 1 <-> WcState/InputToggle
//     Enc/Inputs/In/nState4 <-> WcState/WcState
//     Enc/Outputs/Out/nCtrl1 @bit 3 <-> ENC Control compact/Control/Enable latch extern on negative edge
//     Enc/Outputs/Out/nCtrl1 @bit 1 <-> ENC Control compact/Control/Enable latch extern on positive edge
//     Enc/Outputs/Out/nCtrl1 @bit 2 <-> ENC Control compact/Control/Set counter
//     Enc/Outputs/Out/nDataOut1[0] <-> ENC Control compact/Set counter value
//   tmo_optics Instance <-> Device 1 (EtherCAT)/Term 1 (EK1200)/PMPS_FFO
//     PlcTask Outputs/GVL_PMPS.g_FastFaultOutput1.q_xFastFaultOut <-> Channel 1/Output
//     PlcTask Outputs/GVL_PMPS.g_FastFaultOutput2.q_xFastFaultOut <-> Channel 2/Output
//   tmo_optics Instance <-> Device 1 (EtherCAT)/Term 1 (EK1200)/PMPS_PRE
//     PlcTask Inputs/PRG_PMPS.fbArbiterIO.i_stCurrentBP <-> IO Inputs/CurrentBP
//     PlcTask Inputs/PRG_PMPS.fbArbiterIO.xTxPDO_state <-> SYNC Inputs/TxPDO state
//     PlcTask Inputs/PRG_PMPS.fbArbiterIO.xTxPDO_toggle <-> SYNC Inputs/TxPDO toggle
//     PlcTask Outputs/PRG_PMPS.fbArbiterIO.q_stRequestedBP <-> IO Outputs/RequestedBP
//   tmo_optics Instance <-> Device 1 (EtherCAT)/Term 1 (EK1200)/Term 39 (EK1122)/B940-009-R19-DRL-04 (EK1100)/SL2K4-EL5072-E1
//     PlcTask Inputs/Main.M25.nRawEncoderDINT <-> IND Inputs Channel 1/Position
//     PlcTask Inputs/Main.M26.nRawEncoderDINT <-> IND Inputs Channel 2/Position
//   tmo_optics Instance <-> Device 1 (EtherCAT)/Term 1 (EK1200)/Term 39 (EK1122)/B940-009-R19-DRL-04 (EK1100)/SL2K4-EL5072-E2
//     PlcTask Inputs/Main.M27.nRawEncoderDINT <-> IND Inputs Channel 1/Position
//     PlcTask Inputs/Main.M28.nRawEncoderDINT <-> IND Inputs Channel 2/Position
//   tmo_optics Instance <-> Device 1 (EtherCAT)/Term 1 (EK1200)/Term 39 (EK1122)/Term 110 (EK1100)/EL3054_FWM_PRSM_MR45K4
//     PlcTask Inputs/PRG_MR4K4_KBO.fbCoolingPanel.fbFlow_1.iRaw <-> AI Standard Channel 1/Value
//     PlcTask Inputs/PRG_MR5K4_KBO.fbCoolingPanel.fbFlow_1.iRaw <-> AI Standard Channel 3/Value
//     PlcTask Inputs/PRG_MR4K4_KBO.fbCoolingPanel.fbPress_1.iRaw <-> AI Standard Channel 2/Value
//     PlcTask Inputs/PRG_MR5K4_KBO.fbCoolingPanel.fbPress_1.iRaw <-> AI Standard Channel 2/Value
//   tmo_optics Instance <-> Device 1 (EtherCAT)/Term 1 (EK1200)/Term 39 (EK1122)/Term 110 (EK1100)/EL3204_M4K4
//     PlcTask Inputs/GVL_M4K4_RTD.nM4K4_Chin_Left_RTD.bError <-> RTD Inputs Channel 1/Status/Error
//     PlcTask Inputs/GVL_M4K4_RTD.nM4K4_Chin_Left_RTD.bOverrange <-> RTD Inputs Channel 1/Status/Overrange
//     PlcTask Inputs/GVL_M4K4_RTD.nM4K4_Chin_Left_RTD.bUnderrange <-> RTD Inputs Channel 1/Status/Underrange
//     PlcTask Inputs/GVL_M4K4_RTD.nM4K4_Chin_Left_RTD.iRaw <-> RTD Inputs Channel 1/Value
//     PlcTask Inputs/GVL_M4K4_RTD.nM4K4_Chin_Right_RTD.bError <-> RTD Inputs Channel 2/Status/Error
//     PlcTask Inputs/GVL_M4K4_RTD.nM4K4_Chin_Right_RTD.bOverrange <-> RTD Inputs Channel 2/Status/Overrange
//     PlcTask Inputs/GVL_M4K4_RTD.nM4K4_Chin_Right_RTD.bUnderrange <-> RTD Inputs Channel 2/Status/Underrange
//     PlcTask Inputs/GVL_M4K4_RTD.nM4K4_Chin_Right_RTD.iRaw <-> RTD Inputs Channel 2/Value
//     PlcTask Inputs/GVL_M4K4_RTD.nM4K4_Chin_Tail_RTD.bError <-> RTD Inputs Channel 3/Status/Error
//     PlcTask Inputs/GVL_M4K4_RTD.nM4K4_Chin_Tail_RTD.bOverrange <-> RTD Inputs Channel 3/Status/Overrange
//     PlcTask Inputs/GVL_M4K4_RTD.nM4K4_Chin_Tail_RTD.bUnderrange <-> RTD Inputs Channel 3/Status/Underrange
//     PlcTask Inputs/GVL_M4K4_RTD.nM4K4_Chin_Tail_RTD.iRaw <-> RTD Inputs Channel 3/Value
//   tmo_optics Instance <-> Device 1 (EtherCAT)/Term 1 (EK1200)/Term 39 (EK1122)/Term 110 (EK1100)/EL3204_M5K4
//     PlcTask Inputs/GVL_M5K4_RTD.nM5K4_Chin_Left_RTD.bError <-> RTD Inputs Channel 1/Status/Error
//     PlcTask Inputs/GVL_M5K4_RTD.nM5K4_Chin_Left_RTD.bOverrange <-> RTD Inputs Channel 1/Status/Overrange
//     PlcTask Inputs/GVL_M5K4_RTD.nM5K4_Chin_Left_RTD.bUnderrange <-> RTD Inputs Channel 1/Status/Underrange
//     PlcTask Inputs/GVL_M5K4_RTD.nM5K4_Chin_Left_RTD.iRaw <-> RTD Inputs Channel 1/Value
//     PlcTask Inputs/GVL_M5K4_RTD.nM5K4_Chin_Right_RTD.bError <-> RTD Inputs Channel 2/Status/Error
//     PlcTask Inputs/GVL_M5K4_RTD.nM5K4_Chin_Right_RTD.bOverrange <-> RTD Inputs Channel 2/Status/Overrange
//     PlcTask Inputs/GVL_M5K4_RTD.nM5K4_Chin_Right_RTD.bUnderrange <-> RTD Inputs Channel 2/Status/Underrange
//     PlcTask Inputs/GVL_M5K4_RTD.nM5K4_Chin_Right_RTD.iRaw <-> RTD Inputs Channel 2/Value
//     PlcTask Inputs/GVL_M5K4_RTD.nM5K4_Chin_Tail_RTD.bError <-> RTD Inputs Channel 3/Status/Error
//     PlcTask Inputs/GVL_M5K4_RTD.nM5K4_Chin_Tail_RTD.bOverrange <-> RTD Inputs Channel 3/Status/Overrange
//     PlcTask Inputs/GVL_M5K4_RTD.nM5K4_Chin_Tail_RTD.bUnderrange <-> RTD Inputs Channel 3/Status/Underrange
//     PlcTask Inputs/GVL_M5K4_RTD.nM5K4_Chin_Tail_RTD.iRaw <-> RTD Inputs Channel 3/Value
//   tmo_optics Instance <-> Device 1 (EtherCAT)/Term 1 (EK1200)/Term 39 (EK1122)/Term 94 (EK1100)/EL5042_M4K4X_M4K4Y
//     PlcTask Inputs/Main.M17.nRawEncoderULINT <-> FB Inputs Channel 1/Position
//     PlcTask Inputs/Main.M18.nRawEncoderULINT <-> FB Inputs Channel 2/Position
//   tmo_optics Instance <-> Device 1 (EtherCAT)/Term 1 (EK1200)/Term 39 (EK1122)/Term 94 (EK1100)/EL5042_M4K4Z_M4K4rX
//     PlcTask Inputs/Main.M19.nRawEncoderULINT <-> FB Inputs Channel 1/Position
//     PlcTask Inputs/Main.M20.nRawEncoderULINT <-> FB Inputs Channel 2/Position
//   tmo_optics Instance <-> Device 1 (EtherCAT)/Term 1 (EK1200)/Term 39 (EK1122)/Term 94 (EK1100)/EL5042_M5K4X_M5K4Y
//     PlcTask Inputs/Main.M21.nRawEncoderULINT <-> FB Inputs Channel 1/Position
//     PlcTask Inputs/Main.M22.nRawEncoderULINT <-> FB Inputs Channel 2/Position
//   tmo_optics Instance <-> Device 1 (EtherCAT)/Term 1 (EK1200)/Term 39 (EK1122)/Term 94 (EK1100)/EL5042_M5K4Z_M5K4rY
//     PlcTask Inputs/Main.M23.nRawEncoderULINT <-> FB Inputs Channel 1/Position
//     PlcTask Inputs/Main.M24.nRawEncoderULINT <-> FB Inputs Channel 2/Position
//   tmo_optics Instance <-> Device 1 (EtherCAT)/Term 1 (EK1200)/Term 39 (EK1122)/Term 94 (EK1100)/EL7041-0052_M4K4X
//     PlcTask Inputs/Main.M17.bLimitBackwardEnable <-> STM Status/Status/Digital input 2
//     PlcTask Inputs/Main.M17.bLimitForwardEnable <-> STM Status/Status/Digital input 1
//   tmo_optics Instance <-> Device 1 (EtherCAT)/Term 1 (EK1200)/Term 39 (EK1122)/Term 94 (EK1100)/EL7041-0052_M4K4Y
//     PlcTask Inputs/Main.M18.bLimitBackwardEnable <-> STM Status/Status/Digital input 2
//     PlcTask Inputs/Main.M18.bLimitForwardEnable <-> STM Status/Status/Digital input 1
//   tmo_optics Instance <-> Device 1 (EtherCAT)/Term 1 (EK1200)/Term 39 (EK1122)/Term 94 (EK1100)/EL7041-0052_M4K4Z
//     PlcTask Inputs/Main.M19.bLimitBackwardEnable <-> STM Status/Status/Digital input 1
//     PlcTask Inputs/Main.M19.bLimitForwardEnable <-> STM Status/Status/Digital input 2
//   tmo_optics Instance <-> Device 1 (EtherCAT)/Term 1 (EK1200)/Term 39 (EK1122)/Term 94 (EK1100)/EL7041-0052_M4K4rX
//     PlcTask Inputs/Main.M20.bLimitBackwardEnable <-> STM Status/Status/Digital input 2
//     PlcTask Inputs/Main.M20.bLimitForwardEnable <-> STM Status/Status/Digital input 1
//   tmo_optics Instance <-> Device 1 (EtherCAT)/Term 1 (EK1200)/Term 39 (EK1122)/Term 94 (EK1100)/EL7041-0052_M5K4X
//     PlcTask Inputs/Main.M21.bLimitBackwardEnable <-> STM Status/Status/Digital input 2
//     PlcTask Inputs/Main.M21.bLimitForwardEnable <-> STM Status/Status/Digital input 1
//   tmo_optics Instance <-> Device 1 (EtherCAT)/Term 1 (EK1200)/Term 39 (EK1122)/Term 94 (EK1100)/EL7041-0052_M5K4Y
//     PlcTask Inputs/Main.M22.bLimitBackwardEnable <-> STM Status/Status/Digital input 2
//     PlcTask Inputs/Main.M22.bLimitForwardEnable <-> STM Status/Status/Digital input 1
//   tmo_optics Instance <-> Device 1 (EtherCAT)/Term 1 (EK1200)/Term 39 (EK1122)/Term 94 (EK1100)/EL7041-0052_M5K4Z
//     PlcTask Inputs/Main.M23.bLimitBackwardEnable <-> STM Status/Status/Digital input 1
//     PlcTask Inputs/Main.M23.bLimitForwardEnable <-> STM Status/Status/Digital input 2
//   tmo_optics Instance <-> Device 1 (EtherCAT)/Term 1 (EK1200)/Term 39 (EK1122)/Term 94 (EK1100)/EL7041-0052_M5K4rY
//     PlcTask Inputs/Main.M24.bLimitBackwardEnable <-> STM Status/Status/Digital input 2
//     PlcTask Inputs/Main.M24.bLimitForwardEnable <-> STM Status/Status/Digital input 1
//   tmo_optics Instance <-> Device 1 (EtherCAT)/Term 1 (EK1200)/Term 39 (EK1122)/Term 94 (EK1100)/Term 109 (EL1004)
//     PlcTask Inputs/Main.bDreamEnable1 <-> Channel 1/Input
//     PlcTask Inputs/Main.bDreamEnable2 <-> Channel 2/Input
//   tmo_optics Instance <-> Device 1 (EtherCAT)/Term 1 (EK1200)/Term 5 (EK1122)/EP2008-0001_M1K4_VCV
//     PlcTask Outputs/PRG_MR1K4_SOMS.bActivateVarCool <-> Channel 1/Output
//   tmo_optics Instance <-> Device 1 (EtherCAT)/Term 1 (EK1200)/Term 5 (EK1122)/Term 20 (EK1100)/EL1004_M2K4_M3K4_STO
//     PlcTask Inputs/Main.LAMPbSTOEnable1 <-> Channel 1/Input
//     PlcTask Inputs/Main.LAMPbSTOEnable2 <-> Channel 2/Input
//   tmo_optics Instance <-> Device 1 (EtherCAT)/Term 1 (EK1200)/Term 5 (EK1122)/Term 20 (EK1100)/EL5042_M2K4X_M2K4Y
//     PlcTask Inputs/Main.M7.nRawEncoderULINT <-> FB Inputs Channel 1/Position
//     PlcTask Inputs/Main.M8.nRawEncoderULINT <-> FB Inputs Channel 2/Position
//   tmo_optics Instance <-> Device 1 (EtherCAT)/Term 1 (EK1200)/Term 5 (EK1122)/Term 20 (EK1100)/EL5042_M2K4_BEND_USDS
//     PlcTask Inputs/Main.M10.nRawEncoderULINT <-> FB Inputs Channel 1/Position
//     PlcTask Inputs/Main.M11.nRawEncoderULINT <-> FB Inputs Channel 2/Position
//     PlcTask Inputs/Main.M16.nRawEncoderULINT <-> FB Inputs Channel 2/Position
//   tmo_optics Instance <-> Device 1 (EtherCAT)/Term 1 (EK1200)/Term 5 (EK1122)/Term 20 (EK1100)/EL5042_M2K4rY_M3K4X
//     PlcTask Inputs/Main.M12.nRawEncoderULINT <-> FB Inputs Channel 2/Position
//     PlcTask Inputs/Main.M9.nRawEncoderULINT <-> FB Inputs Channel 1/Position
//   tmo_optics Instance <-> Device 1 (EtherCAT)/Term 1 (EK1200)/Term 5 (EK1122)/Term 20 (EK1100)/EL5042_M3K4Y_M3K4rX
//     PlcTask Inputs/Main.M13.nRawEncoderULINT <-> FB Inputs Channel 1/Position
//     PlcTask Inputs/Main.M14.nRawEncoderULINT <-> FB Inputs Channel 2/Position
//   tmo_optics Instance <-> Device 1 (EtherCAT)/Term 1 (EK1200)/Term 5 (EK1122)/Term 20 (EK1100)/EL5042_M3K4_BEND_USDS
//     PlcTask Inputs/Main.M15.nRawEncoderULINT <-> FB Inputs Channel 1/Position
//   tmo_optics Instance <-> Device 1 (EtherCAT)/Term 1 (EK1200)/Term 5 (EK1122)/Term 20 (EK1100)/EL7041-0052_M2K4X
//     PlcTask Inputs/Main.M7.bLimitBackwardEnable <-> STM Status/Status/Digital input 2
//     PlcTask Inputs/Main.M7.bLimitForwardEnable <-> STM Status/Status/Digital input 1
//   tmo_optics Instance <-> Device 1 (EtherCAT)/Term 1 (EK1200)/Term 5 (EK1122)/Term 20 (EK1100)/EL7041-0052_M2K4Y
//     PlcTask Inputs/Main.M8.bLimitBackwardEnable <-> STM Status/Status/Digital input 2
//     PlcTask Inputs/Main.M8.bLimitForwardEnable <-> STM Status/Status/Digital input 1
//   tmo_optics Instance <-> Device 1 (EtherCAT)/Term 1 (EK1200)/Term 5 (EK1122)/Term 20 (EK1100)/EL7041-0052_M2K4rY
//     PlcTask Inputs/Main.M9.bLimitBackwardEnable <-> STM Status/Status/Digital input 2
//     PlcTask Inputs/Main.M9.bLimitForwardEnable <-> STM Status/Status/Digital input 1
//   tmo_optics Instance <-> Device 1 (EtherCAT)/Term 1 (EK1200)/Term 5 (EK1122)/Term 20 (EK1100)/EL7041-0052_M3K4X
//     PlcTask Inputs/Main.M12.bLimitBackwardEnable <-> STM Status/Status/Digital input 2
//     PlcTask Inputs/Main.M12.bLimitForwardEnable <-> STM Status/Status/Digital input 1
//   tmo_optics Instance <-> Device 1 (EtherCAT)/Term 1 (EK1200)/Term 5 (EK1122)/Term 20 (EK1100)/EL7041-0052_M3K4Y
//     PlcTask Inputs/Main.M13.bLimitBackwardEnable <-> STM Status/Status/Digital input 2
//     PlcTask Inputs/Main.M13.bLimitForwardEnable <-> STM Status/Status/Digital input 1
//   tmo_optics Instance <-> Device 1 (EtherCAT)/Term 1 (EK1200)/Term 5 (EK1122)/Term 20 (EK1100)/EL7041-0052_M3K4rX
//     PlcTask Inputs/Main.M14.bLimitBackwardEnable <-> STM Status/Status/Digital input 2
//     PlcTask Inputs/Main.M14.bLimitForwardEnable <-> STM Status/Status/Digital input 1
//   tmo_optics Instance <-> Device 1 (EtherCAT)/Term 1 (EK1200)/Term 5 (EK1122)/Term 20 (EK1100)/EL7041_M2K4_BEND_DS
//     PlcTask Inputs/Main.M11.bLimitBackwardEnable <-> STM Status/Status/Digital input 2
//     PlcTask Inputs/Main.M11.bLimitForwardEnable <-> STM Status/Status/Digital input 1
//   tmo_optics Instance <-> Device 1 (EtherCAT)/Term 1 (EK1200)/Term 5 (EK1122)/Term 20 (EK1100)/EL7041_M2K4_BEND_US
//     PlcTask Inputs/Main.M10.bLimitBackwardEnable <-> STM Status/Status/Digital input 2
//     PlcTask Inputs/Main.M10.bLimitForwardEnable <-> STM Status/Status/Digital input 1
//   tmo_optics Instance <-> Device 1 (EtherCAT)/Term 1 (EK1200)/Term 5 (EK1122)/Term 20 (EK1100)/EL7041_M3K4_BEND_DS
//     PlcTask Inputs/Main.M16.bLimitBackwardEnable <-> STM Status/Status/Digital input 2
//     PlcTask Inputs/Main.M16.bLimitForwardEnable <-> STM Status/Status/Digital input 1
//   tmo_optics Instance <-> Device 1 (EtherCAT)/Term 1 (EK1200)/Term 5 (EK1122)/Term 20 (EK1100)/EL7041_M3K4_BEND_US
//     PlcTask Inputs/Main.M15.bLimitBackwardEnable <-> STM Status/Status/Digital input 2
//     PlcTask Inputs/Main.M15.bLimitForwardEnable <-> STM Status/Status/Digital input 1
//   tmo_optics Instance <-> Device 1 (EtherCAT)/Term 1 (EK1200)/Term 5 (EK1122)/Term 40 (EK1100)/EL3054_FWM_PRSM
//     PlcTask Inputs/PRG_MR2K4_KBO.fbCoolingPanel.fbFlow_1.iRaw <-> AI Standard Channel 1/Value
//     PlcTask Inputs/PRG_MR3K4_KBO.fbCoolingPanel.fbFlow_1.iRaw <-> AI Standard Channel 2/Value
//     PlcTask Inputs/PRG_MR2K4_KBO.fbCoolingPanel.fbPress_1.iRaw <-> AI Standard Channel 3/Value
//     PlcTask Inputs/PRG_MR3K4_KBO.fbCoolingPanel.fbPress_1.iRaw <-> AI Standard Channel 3/Value
//   tmo_optics Instance <-> Device 1 (EtherCAT)/Term 1 (EK1200)/Term 5 (EK1122)/Term 40 (EK1100)/EL3202-0010_M2K4DS2_M2K4DS3
//     PlcTask Inputs/GVL_M2K4_RTD.nM2K4DS_RTD_3 <-> RTD Inputs Channel 2/Value
//     PlcTask Inputs/PRG_MR2K4_KBO.fbM2K4_Chin_Right_RTD.bError <-> RTD Inputs Channel 1/Status/Error
//     PlcTask Inputs/PRG_MR2K4_KBO.fbM2K4_Chin_Right_RTD.bOverrange <-> RTD Inputs Channel 1/Status/Overrange
//     PlcTask Inputs/PRG_MR2K4_KBO.fbM2K4_Chin_Right_RTD.bUnderrange <-> RTD Inputs Channel 1/Status/Underrange
//     PlcTask Inputs/PRG_MR2K4_KBO.fbM2K4_Chin_Right_RTD.iRaw <-> RTD Inputs Channel 1/Value
//     PlcTask Inputs/P_StripeProtections.fbStripProtMR2K4.ffLowerCoatingRTemp.bError <-> RTD Inputs Channel 1/Status/Error
//     PlcTask Inputs/P_StripeProtections.fbStripProtMR2K4.ffLowerCoatingRTemp.bOverrange <-> RTD Inputs Channel 1/Status/Overrange
//     PlcTask Inputs/P_StripeProtections.fbStripProtMR2K4.ffLowerCoatingRTemp.bUnderrange <-> RTD Inputs Channel 1/Status/Underrange
//     PlcTask Inputs/P_StripeProtections.fbStripProtMR2K4.ffLowerCoatingRTemp.iRaw <-> RTD Inputs Channel 1/Value
//     PlcTask Inputs/P_StripeProtections.fbStripProtMR2K4.ffUpperCoatingRTemp.bError <-> RTD Inputs Channel 1/Status/Error
//     PlcTask Inputs/P_StripeProtections.fbStripProtMR2K4.ffUpperCoatingRTemp.bOverrange <-> RTD Inputs Channel 1/Status/Overrange
//     PlcTask Inputs/P_StripeProtections.fbStripProtMR2K4.ffUpperCoatingRTemp.bUnderrange <-> RTD Inputs Channel 1/Status/Underrange
//     PlcTask Inputs/P_StripeProtections.fbStripProtMR2K4.ffUpperCoatingRTemp.iRaw <-> RTD Inputs Channel 1/Value
//   tmo_optics Instance <-> Device 1 (EtherCAT)/Term 1 (EK1200)/Term 5 (EK1122)/Term 40 (EK1100)/EL3202-0010_M2K4US1_M2K4US2
//     PlcTask Inputs/GVL_M2K4_RTD.nM2K4US_RTD_1 <-> RTD Inputs Channel 1/Value
//     PlcTask Inputs/PRG_MR2K4_KBO.fbM2K4_Chin_Left_RTD.bError <-> RTD Inputs Channel 2/Status/Error
//     PlcTask Inputs/PRG_MR2K4_KBO.fbM2K4_Chin_Left_RTD.bOverrange <-> RTD Inputs Channel 2/Status/Overrange
//     PlcTask Inputs/PRG_MR2K4_KBO.fbM2K4_Chin_Left_RTD.bUnderrange <-> RTD Inputs Channel 2/Status/Underrange
//     PlcTask Inputs/PRG_MR2K4_KBO.fbM2K4_Chin_Left_RTD.iRaw <-> RTD Inputs Channel 2/Value
//     PlcTask Inputs/P_StripeProtections.fbStripProtMR2K4.ffLowerCoatingLTemp.bError <-> RTD Inputs Channel 2/Status/Error
//     PlcTask Inputs/P_StripeProtections.fbStripProtMR2K4.ffLowerCoatingLTemp.bOverrange <-> RTD Inputs Channel 2/Status/Overrange
//     PlcTask Inputs/P_StripeProtections.fbStripProtMR2K4.ffLowerCoatingLTemp.bUnderrange <-> RTD Inputs Channel 2/Status/Underrange
//     PlcTask Inputs/P_StripeProtections.fbStripProtMR2K4.ffLowerCoatingLTemp.iRaw <-> RTD Inputs Channel 2/Value
//     PlcTask Inputs/P_StripeProtections.fbStripProtMR2K4.ffUpperCoatingLTemp.bError <-> RTD Inputs Channel 2/Status/Error
//     PlcTask Inputs/P_StripeProtections.fbStripProtMR2K4.ffUpperCoatingLTemp.bOverrange <-> RTD Inputs Channel 2/Status/Overrange
//     PlcTask Inputs/P_StripeProtections.fbStripProtMR2K4.ffUpperCoatingLTemp.bUnderrange <-> RTD Inputs Channel 2/Status/Underrange
//     PlcTask Inputs/P_StripeProtections.fbStripProtMR2K4.ffUpperCoatingLTemp.iRaw <-> RTD Inputs Channel 2/Value
//   tmo_optics Instance <-> Device 1 (EtherCAT)/Term 1 (EK1200)/Term 5 (EK1122)/Term 40 (EK1100)/EL3202-0010_M2K4US3_M2K4DS1
//     PlcTask Inputs/GVL_M2K4_RTD.nM2K4DS_RTD_1 <-> RTD Inputs Channel 2/Value
//     PlcTask Inputs/GVL_M2K4_RTD.nM2K4US_RTD_3 <-> RTD Inputs Channel 1/Value
//   tmo_optics Instance <-> Device 1 (EtherCAT)/Term 1 (EK1200)/Term 5 (EK1122)/Term 40 (EK1100)/EL3202-0010_M3K4DS2_M3K4DS3
//     PlcTask Inputs/GVL_M3K4_RTD.nM3K4DS_RTD_3 <-> RTD Inputs Channel 2/Value
//     PlcTask Inputs/PRG_MR3K4_KBO.fbM3K4_Chin_Right_RTD.bError <-> RTD Inputs Channel 1/Status/Error
//     PlcTask Inputs/PRG_MR3K4_KBO.fbM3K4_Chin_Right_RTD.bOverrange <-> RTD Inputs Channel 1/Status/Overrange
//     PlcTask Inputs/PRG_MR3K4_KBO.fbM3K4_Chin_Right_RTD.bUnderrange <-> RTD Inputs Channel 1/Status/Underrange
//     PlcTask Inputs/PRG_MR3K4_KBO.fbM3K4_Chin_Right_RTD.iRaw <-> RTD Inputs Channel 1/Value
//     PlcTask Inputs/P_StripeProtections.fbStripProtMR3K4.ffLowerCoatingRTemp.bError <-> RTD Inputs Channel 1/Status/Error
//     PlcTask Inputs/P_StripeProtections.fbStripProtMR3K4.ffLowerCoatingRTemp.bOverrange <-> RTD Inputs Channel 1/Status/Overrange
//     PlcTask Inputs/P_StripeProtections.fbStripProtMR3K4.ffLowerCoatingRTemp.bUnderrange <-> RTD Inputs Channel 1/Status/Underrange
//     PlcTask Inputs/P_StripeProtections.fbStripProtMR3K4.ffLowerCoatingRTemp.iRaw <-> RTD Inputs Channel 1/Value
//     PlcTask Inputs/P_StripeProtections.fbStripProtMR3K4.ffUpperCoatingRTemp.bError <-> RTD Inputs Channel 1/Status/Error
//     PlcTask Inputs/P_StripeProtections.fbStripProtMR3K4.ffUpperCoatingRTemp.bOverrange <-> RTD Inputs Channel 1/Status/Overrange
//     PlcTask Inputs/P_StripeProtections.fbStripProtMR3K4.ffUpperCoatingRTemp.bUnderrange <-> RTD Inputs Channel 1/Status/Underrange
//     PlcTask Inputs/P_StripeProtections.fbStripProtMR3K4.ffUpperCoatingRTemp.iRaw <-> RTD Inputs Channel 1/Value
//   tmo_optics Instance <-> Device 1 (EtherCAT)/Term 1 (EK1200)/Term 5 (EK1122)/Term 40 (EK1100)/EL3202-0010_M3K4US1_M3K4US2
//     PlcTask Inputs/GVL_M3K4_RTD.nM3K4US_RTD_1 <-> RTD Inputs Channel 1/Value
//     PlcTask Inputs/PRG_MR3K4_KBO.fbM3K4_Chin_Left_RTD.bError <-> RTD Inputs Channel 2/Status/Error
//     PlcTask Inputs/PRG_MR3K4_KBO.fbM3K4_Chin_Left_RTD.bOverrange <-> RTD Inputs Channel 2/Status/Overrange
//     PlcTask Inputs/PRG_MR3K4_KBO.fbM3K4_Chin_Left_RTD.bUnderrange <-> RTD Inputs Channel 2/Status/Underrange
//     PlcTask Inputs/PRG_MR3K4_KBO.fbM3K4_Chin_Left_RTD.iRaw <-> RTD Inputs Channel 2/Value
//     PlcTask Inputs/P_StripeProtections.fbStripProtMR3K4.ffLowerCoatingLTemp.bError <-> RTD Inputs Channel 2/Status/Error
//     PlcTask Inputs/P_StripeProtections.fbStripProtMR3K4.ffLowerCoatingLTemp.bOverrange <-> RTD Inputs Channel 2/Status/Overrange
//     PlcTask Inputs/P_StripeProtections.fbStripProtMR3K4.ffLowerCoatingLTemp.bUnderrange <-> RTD Inputs Channel 2/Status/Underrange
//     PlcTask Inputs/P_StripeProtections.fbStripProtMR3K4.ffLowerCoatingLTemp.iRaw <-> RTD Inputs Channel 2/Value
//     PlcTask Inputs/P_StripeProtections.fbStripProtMR3K4.ffUpperCoatingLTemp.bError <-> RTD Inputs Channel 2/Status/Error
//     PlcTask Inputs/P_StripeProtections.fbStripProtMR3K4.ffUpperCoatingLTemp.bOverrange <-> RTD Inputs Channel 2/Status/Overrange
//     PlcTask Inputs/P_StripeProtections.fbStripProtMR3K4.ffUpperCoatingLTemp.bUnderrange <-> RTD Inputs Channel 2/Status/Underrange
//     PlcTask Inputs/P_StripeProtections.fbStripProtMR3K4.ffUpperCoatingLTemp.iRaw <-> RTD Inputs Channel 2/Value
//   tmo_optics Instance <-> Device 1 (EtherCAT)/Term 1 (EK1200)/Term 5 (EK1122)/Term 40 (EK1100)/EL3202-0010_M3K4US3_M3K4DS1
//     PlcTask Inputs/GVL_M3K4_RTD.nM3K4DS_RTD_1 <-> RTD Inputs Channel 2/Value
//     PlcTask Inputs/GVL_M3K4_RTD.nM3K4US_RTD_3 <-> RTD Inputs Channel 1/Value
//   tmo_optics Instance <-> Device 1 (EtherCAT)/Term 1 (EK1200)/Term 5 (EK1122)/Term 6 (EK1100)/EL1004_M1K4_STO
//     PlcTask Inputs/Main.M1K4.fbRunHOMS.bSTOEnable1 <-> Channel 1/Input
//     PlcTask Inputs/Main.M1K4.fbRunHOMS.bSTOEnable2 <-> Channel 2/Input
//   tmo_optics Instance <-> Device 1 (EtherCAT)/Term 1 (EK1200)/Term 5 (EK1122)/Term 6 (EK1100)/EL3054_M1K4_FWM_PRSM
//     PlcTask Inputs/PRG_MR1K4_SOMS.fbCoolingPanel.fbFlow_1.iRaw <-> AI Standard Channel 1/Value
//     PlcTask Inputs/PRG_MR1K4_SOMS.fbCoolingPanel.fbFlow_2.iRaw <-> AI Standard Channel 2/Value
//     PlcTask Inputs/PRG_MR1K4_SOMS.fbCoolingPanel.fbPress_1.iRaw <-> AI Standard Channel 3/Value
//   tmo_optics Instance <-> Device 1 (EtherCAT)/Term 1 (EK1200)/Term 5 (EK1122)/Term 6 (EK1100)/EL5042_M1K4_PitchBender
//     PlcTask Inputs/GVL_M1K4.M1K4_Pitch.diEncCnt <-> FB Inputs Channel 1/Position
//   tmo_optics Instance <-> Device 1 (EtherCAT)/Term 1 (EK1200)/Term 5 (EK1122)/Term 6 (EK1100)/EL5042_M1K4_Xupdwn
//     PlcTask Inputs/Main.M1K4.fbRunHOMS.stXdwnEnc/Count <-> FB Inputs Channel 2/Position
//     PlcTask Inputs/Main.M1K4.fbRunHOMS.stXupEnc/Count <-> FB Inputs Channel 1/Position
//   tmo_optics Instance <-> Device 1 (EtherCAT)/Term 1 (EK1200)/Term 5 (EK1122)/Term 6 (EK1100)/EL5042_M1K4_Yupdwn
//     PlcTask Inputs/Main.M1K4.fbRunHOMS.stYdwnEnc/Count <-> FB Inputs Channel 2/Position
//     PlcTask Inputs/Main.M1K4.fbRunHOMS.stYupEnc/Count <-> FB Inputs Channel 1/Position
//   tmo_optics Instance <-> Device 1 (EtherCAT)/Term 1 (EK1200)/Term 5 (EK1122)/Term 6 (EK1100)/EL6001_M1K4_PitchFine
//     SerialIO Inputs/GVL_SerialIO.Serial_stComIn_M1K4/D[{0..21}] <-> COM Inputs/Data In {0..21}  (22 links)
//     SerialIO Inputs/GVL_SerialIO.Serial_stComIn_M1K4/Status <-> COM Inputs/Status
//     SerialIO Outputs/GVL_SerialIO.Serial_stComOut_M1K4/Ctrl <-> COM Outputs/Ctrl
//     SerialIO Outputs/GVL_SerialIO.Serial_stComOut_M1K4/D[{0..21}] <-> COM Outputs/Data Out {0..21}  (22 links)
//   tmo_optics Instance <-> Device 1 (EtherCAT)/Term 1 (EK1200)/Term 5 (EK1122)/Term 6 (EK1100)/EL7041-1000_M1K4_PitchCoarse
//     PlcTask Inputs/Main.M5.bLimitBackwardEnable <-> STM Status/Status/Digital input 2
//     PlcTask Inputs/Main.M5.bLimitForwardEnable <-> STM Status/Status/Digital input 1
//   tmo_optics Instance <-> Device 1 (EtherCAT)/Term 1 (EK1200)/Term 5 (EK1122)/Term 6 (EK1100)/EL7041-1000_M1K4_Xdwn
//     PlcTask Inputs/Main.M4.bLimitBackwardEnable <-> STM Status/Status/Digital input 2
//     PlcTask Inputs/Main.M4.bLimitForwardEnable <-> STM Status/Status/Digital input 1
//   tmo_optics Instance <-> Device 1 (EtherCAT)/Term 1 (EK1200)/Term 5 (EK1122)/Term 6 (EK1100)/EL7041-1000_M1K4_Xup
//     PlcTask Inputs/Main.M3.bLimitBackwardEnable <-> STM Status/Status/Digital input 2
//     PlcTask Inputs/Main.M3.bLimitForwardEnable <-> STM Status/Status/Digital input 1
//   tmo_optics Instance <-> Device 1 (EtherCAT)/Term 1 (EK1200)/Term 5 (EK1122)/Term 6 (EK1100)/EL7041-1000_M1K4_Ydwn
//     PlcTask Inputs/Main.M2.bLimitBackwardEnable <-> STM Status/Status/Digital input 2
//     PlcTask Inputs/Main.M2.bLimitForwardEnable <-> STM Status/Status/Digital input 1
//   tmo_optics Instance <-> Device 1 (EtherCAT)/Term 1 (EK1200)/Term 5 (EK1122)/Term 6 (EK1100)/EL7041-1000_M1K4_Yup
//     PlcTask Inputs/Main.M1.bLimitBackwardEnable <-> STM Status/Status/Digital input 2
//     PlcTask Inputs/Main.M1.bLimitForwardEnable <-> STM Status/Status/Digital input 1
//   tmo_optics Instance <-> NC-Task 1 SAF/Axes/M1K4-Pitch
//     PlcTask Inputs/Main.M5.Axis.NcToPlc <-> Outputs/ToPlc
//     PlcTask Outputs/Main.M5.Axis.PlcToNc <-> Inputs/FromPlc
//   tmo_optics Instance <-> NC-Task 1 SAF/Axes/M1K4-Xdwn
//     PlcTask Inputs/Main.M4.Axis.NcToPlc <-> Outputs/ToPlc
//     PlcTask Outputs/Main.M4.Axis.PlcToNc <-> Inputs/FromPlc
//   tmo_optics Instance <-> NC-Task 1 SAF/Axes/M1K4-Xup
